Yaskawa INFORM job: DEMO_ROOF_UPPER_0625_3PAINT_57.JBI

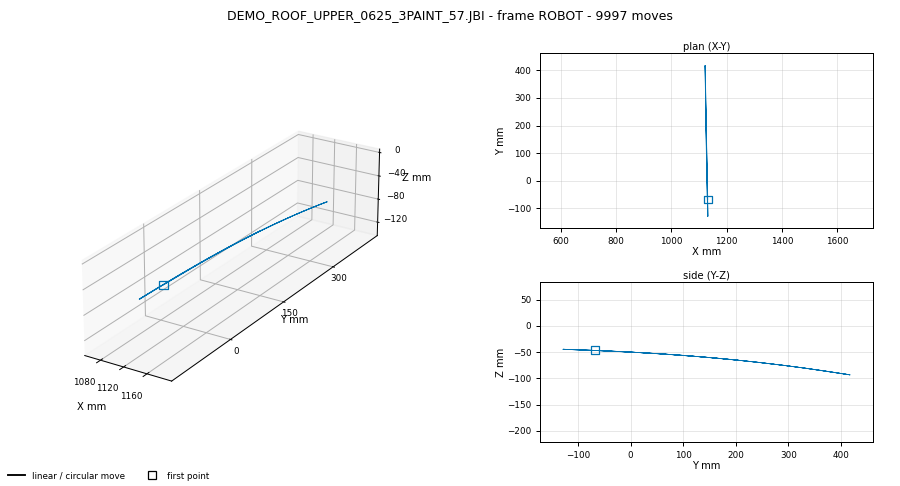
[picture p0: tool path of DEMO_ROOF_UPPER_0625_3PAINT_57.JBI in frame ROBOT, 9997 of 9997 moves have a stored position in this frame; points joined in program order, loops and branches not executed]
/JOB
//NAME DEMO_ROOF_UPPER_0625_3PAINT57
//POS
///NPOS 9997,0,0,0,0,0
///TOOL 0
///USER 0
///POSTYPE ROBOT
///RECTAN
///RCONF 1,0,0,0,0,0,0,0,0,0,0,0,0,0,0,0,0,0,0,0,0,0,0,0
C00000=1131.669,-67.518,-46.703,178.917,6.184,149.436
C00001=1131.665,-67.268,-46.713,178.919,6.185,149.435
C00002=1131.659,-67.019,-46.724,178.922,6.185,149.435
C00003=1131.653,-66.769,-46.734,178.924,6.186,149.434
C00004=1131.648,-66.519,-46.744,178.926,6.187,149.434
C00005=1131.643,-66.269,-46.754,178.928,6.187,149.433
C00006=1131.637,-66.020,-46.765,178.930,6.188,149.433
C00007=1131.632,-65.770,-46.775,178.932,6.188,149.432
C00008=1131.627,-65.520,-46.785,178.935,6.189,149.432
C00009=1131.622,-65.271,-46.795,178.937,6.189,149.431
C00010=1131.617,-65.021,-46.806,178.939,6.190,149.431
C00011=1131.611,-64.771,-46.816,178.941,6.190,149.430
C00012=1131.606,-64.521,-46.826,178.943,6.191,149.429
C00013=1131.601,-64.271,-46.837,178.946,6.191,149.429
C00014=1131.595,-64.022,-46.847,178.948,6.192,149.428
C00015=1131.590,-63.772,-46.858,178.950,6.193,149.428
C00016=1131.585,-63.522,-46.868,178.952,6.194,149.427
C00017=1131.579,-63.273,-46.879,178.955,6.194,149.427
C00018=1131.574,-63.023,-46.889,178.956,6.194,149.426
C00019=1131.568,-62.773,-46.899,178.959,6.195,149.426
C00020=1131.563,-62.524,-46.910,178.961,6.195,149.425
C00021=1131.558,-62.273,-46.920,178.963,6.196,149.425
C00022=1131.552,-62.024,-46.930,178.966,6.197,149.424
C00023=1131.548,-61.774,-46.940,178.968,6.197,149.424
C00024=1131.543,-61.525,-46.951,178.970,6.198,149.423
C00025=1131.537,-61.275,-46.961,178.972,6.198,149.423
C00026=1131.532,-61.025,-46.972,178.974,6.199,149.422
C00027=1131.527,-60.776,-46.982,178.976,6.199,149.421
C00028=1131.522,-60.525,-46.993,178.979,6.200,149.421
C00029=1131.516,-60.276,-47.004,178.981,6.201,149.421
C00030=1131.511,-60.026,-47.014,178.983,6.202,149.420
C00031=1131.506,-59.777,-47.025,178.985,6.202,149.420
C00032=1131.500,-59.527,-47.035,178.987,6.202,149.419
C00033=1131.495,-59.277,-47.045,178.989,6.203,149.418
C00034=1131.490,-59.028,-47.056,178.992,6.203,149.418
C00035=1131.485,-58.778,-47.067,178.994,6.204,149.417
C00036=1131.479,-58.528,-47.077,178.997,6.205,149.417
C00037=1131.474,-58.278,-47.088,178.999,6.205,149.416
C00038=1131.468,-58.029,-47.099,179.001,6.206,149.416
C00039=1131.463,-57.778,-47.110,179.003,6.207,149.415
C00040=1131.458,-57.529,-47.120,179.005,6.208,149.415
C00041=1131.453,-57.279,-47.130,179.007,6.207,149.414
C00042=1131.447,-57.030,-47.141,179.010,6.208,149.414
C00043=1131.442,-56.780,-47.152,179.012,6.209,149.413
C00044=1131.437,-56.530,-47.162,179.014,6.210,149.413
C00045=1131.431,-56.280,-47.172,179.016,6.210,149.412
C00046=1131.426,-56.031,-47.184,179.019,6.211,149.411
C00047=1131.421,-55.781,-47.194,179.021,6.211,149.411
C00048=1131.416,-55.531,-47.204,179.023,6.212,149.410
C00049=1131.410,-55.282,-47.215,179.025,6.213,149.410
C00050=1131.405,-55.032,-47.226,179.027,6.213,149.409
C00051=1131.400,-54.782,-47.236,179.030,6.213,149.409
C00052=1131.394,-54.532,-47.248,179.032,6.214,149.408
C00053=1131.389,-54.283,-47.258,179.034,6.215,149.408
C00054=1131.384,-54.033,-47.270,179.036,6.216,149.407
C00055=1131.379,-53.784,-47.280,179.039,6.216,149.407
C00056=1131.374,-53.533,-47.290,179.041,6.217,149.406
C00057=1131.369,-53.284,-47.302,179.043,6.218,149.406
C00058=1131.363,-53.034,-47.312,179.045,6.218,149.405
C00059=1131.358,-52.784,-47.324,179.048,6.219,149.405
C00060=1131.352,-52.535,-47.334,179.050,6.219,149.404
C00061=1131.347,-52.284,-47.345,179.052,6.219,149.404
C00062=1131.342,-52.036,-47.355,179.054,6.220,149.403
C00063=1131.337,-51.785,-47.366,179.057,6.221,149.402
C00064=1131.332,-51.536,-47.377,179.059,6.221,149.402
C00065=1131.326,-51.265,-47.388,179.061,6.222,149.401
C00066=1131.320,-50.994,-47.401,179.064,6.222,149.401
C00067=1131.314,-50.724,-47.413,179.066,6.223,149.400
C00068=1131.309,-50.453,-47.424,179.069,6.225,149.400
C00069=1131.303,-50.203,-47.435,179.071,6.224,149.399
C00070=1131.298,-49.953,-47.446,179.073,6.225,149.399
C00071=1131.293,-49.703,-47.457,179.075,6.226,149.398
C00072=1131.288,-49.454,-47.468,179.077,6.227,149.398
C00073=1131.282,-49.204,-47.479,179.080,6.227,149.397
C00074=1131.277,-48.955,-47.490,179.082,6.228,149.396
C00075=1131.272,-48.704,-47.501,179.084,6.229,149.396
C00076=1131.266,-48.456,-47.511,179.087,6.229,149.396
C00077=1131.261,-48.205,-47.523,179.089,6.230,149.395
C00078=1131.256,-47.955,-47.534,179.092,6.231,149.394
C00079=1131.250,-47.706,-47.544,179.094,6.231,149.394
C00080=1131.246,-47.456,-47.555,179.096,6.232,149.393
C00081=1131.240,-47.207,-47.567,179.099,6.232,149.393
C00082=1131.235,-46.957,-47.577,179.101,6.233,149.392
C00083=1131.230,-46.707,-47.589,179.103,6.234,149.392
C00084=1131.224,-46.457,-47.600,179.105,6.235,149.391
C00085=1131.219,-46.208,-47.611,179.108,6.235,149.391
C00086=1131.214,-45.958,-47.622,179.110,6.236,149.390
C00087=1131.208,-45.708,-47.633,179.112,6.236,149.390
C00088=1131.203,-45.459,-47.644,179.114,6.237,149.389
C00089=1131.198,-45.209,-47.654,179.116,6.237,149.388
C00090=1131.192,-44.959,-47.666,179.119,6.238,149.388
C00091=1131.188,-44.709,-47.678,179.121,6.239,149.387
C00092=1131.182,-44.460,-47.688,179.123,6.239,149.387
C00093=1131.176,-44.210,-47.700,179.126,6.240,149.386
C00094=1131.172,-43.960,-47.711,179.128,6.241,149.386
C00095=1131.166,-43.711,-47.721,179.130,6.241,149.385
C00096=1131.161,-43.461,-47.733,179.132,6.242,149.385
C00097=1131.156,-43.211,-47.744,179.135,6.243,149.384
C00098=1131.151,-42.962,-47.755,179.137,6.243,149.384
C00099=1131.145,-42.712,-47.767,179.139,6.244,149.383
C00100=1131.140,-42.462,-47.778,179.141,6.245,149.383
C00101=1131.134,-42.213,-47.789,179.144,6.245,149.382
C00102=1131.130,-41.963,-47.801,179.146,6.246,149.382
C00103=1131.125,-41.713,-47.811,179.149,6.247,149.381
C00104=1131.119,-41.463,-47.823,179.151,6.248,149.381
C00105=1131.114,-41.214,-47.834,179.153,6.248,149.380
C00106=1131.108,-40.964,-47.846,179.156,6.249,149.379
C00107=1131.103,-40.714,-47.856,179.158,6.249,149.379
C00108=1131.098,-40.465,-47.867,179.160,6.250,149.378
C00109=1131.093,-40.215,-47.879,179.163,6.251,149.378
C00110=1131.088,-39.965,-47.891,179.165,6.251,149.377
C00111=1131.082,-39.716,-47.902,179.167,6.252,149.377
C00112=1131.077,-39.466,-47.913,179.169,6.253,149.376
C00113=1131.072,-39.216,-47.925,179.172,6.253,149.376
C00114=1131.067,-38.966,-47.936,179.174,6.254,149.375
C00115=1131.061,-38.717,-47.947,179.176,6.255,149.375
C00116=1131.056,-38.468,-47.959,179.178,6.256,149.374
C00117=1131.051,-38.218,-47.971,179.181,6.256,149.373
C00118=1131.046,-37.967,-47.981,179.183,6.257,149.373
C00119=1131.040,-37.718,-47.993,179.185,6.258,149.373
C00120=1131.035,-37.469,-48.004,179.188,6.258,149.372
C00121=1131.030,-37.219,-48.016,179.190,6.259,149.371
C00122=1131.025,-36.969,-48.027,179.192,6.260,149.371
C00123=1131.019,-36.720,-48.039,179.195,6.260,149.370
C00124=1131.014,-36.470,-48.050,179.197,6.261,149.370
C00125=1131.009,-36.220,-48.062,179.200,6.262,149.369
C00126=1131.004,-35.971,-48.073,179.202,6.262,149.369
C00127=1130.998,-35.721,-48.085,179.204,6.263,149.368
C00128=1130.993,-35.471,-48.095,179.207,6.263,149.368
C00129=1130.988,-35.221,-48.107,179.209,6.264,149.367
C00130=1130.982,-34.971,-48.119,179.211,6.265,149.367
C00131=1130.977,-34.722,-48.130,179.213,6.266,149.366
C00132=1130.971,-34.472,-48.142,179.216,6.266,149.365
C00133=1130.967,-34.223,-48.153,179.218,6.267,149.365
C00134=1130.961,-33.973,-48.165,179.220,6.268,149.364
C00135=1130.957,-33.723,-48.176,179.223,6.268,149.364
C00136=1130.951,-33.473,-48.188,179.225,6.269,149.363
C00137=1130.945,-33.224,-48.200,179.227,6.270,149.363
C00138=1130.941,-32.974,-48.211,179.229,6.270,149.362
C00139=1130.935,-32.724,-48.223,179.232,6.271,149.362
C00140=1130.930,-32.475,-48.234,179.234,6.272,149.361
C00141=1130.925,-32.225,-48.246,179.236,6.272,149.361
C00142=1130.920,-31.975,-48.258,179.239,6.273,149.360
C00143=1130.915,-31.727,-48.269,179.242,6.274,149.360
C00144=1130.909,-31.477,-48.281,179.244,6.275,149.359
C00145=1130.904,-31.227,-48.293,179.246,6.276,149.359
C00146=1130.899,-30.977,-48.305,179.249,6.276,149.358
C00147=1130.894,-30.727,-48.316,179.251,6.277,149.357
C00148=1130.888,-30.477,-48.328,179.253,6.278,149.357
C00149=1130.883,-30.228,-48.340,179.255,6.279,149.356
C00150=1130.878,-29.978,-48.351,179.258,6.279,149.356
C00151=1130.872,-29.728,-48.363,179.260,6.280,149.355
C00152=1130.868,-29.479,-48.375,179.263,6.281,149.355
C00153=1130.862,-29.229,-48.387,179.265,6.281,149.354
C00154=1130.857,-28.980,-48.399,179.267,6.282,149.354
C00155=1130.852,-28.730,-48.410,179.270,6.283,149.353
C00156=1130.847,-28.480,-48.422,179.272,6.283,149.353
C00157=1130.841,-28.230,-48.434,179.274,6.284,149.352
C00158=1130.836,-27.980,-48.445,179.277,6.285,149.352
C00159=1130.831,-27.731,-48.458,179.279,6.285,149.351
C00160=1130.825,-27.482,-48.469,179.282,6.287,149.351
C00161=1130.820,-27.232,-48.481,179.284,6.287,149.350
C00162=1130.815,-26.982,-48.492,179.286,6.288,149.349
C00163=1130.810,-26.733,-48.505,179.289,6.289,149.349
C00164=1130.805,-26.483,-48.517,179.291,6.289,149.348
C00165=1130.800,-26.233,-48.528,179.293,6.290,149.348
C00166=1130.795,-25.983,-48.540,179.296,6.291,149.347
C00167=1130.789,-25.734,-48.553,179.298,6.292,149.347
C00168=1130.784,-25.484,-48.565,179.300,6.292,149.346
C00169=1130.779,-25.214,-48.578,179.303,6.293,149.346
C00170=1130.773,-24.944,-48.590,179.306,6.294,149.345
C00171=1130.767,-24.674,-48.603,179.308,6.295,149.344
C00172=1130.762,-24.404,-48.616,179.311,6.295,149.344
C00173=1130.756,-24.154,-48.628,179.313,6.296,149.343
C00174=1130.751,-23.904,-48.639,179.315,6.297,149.343
C00175=1130.746,-23.655,-48.652,179.318,6.297,149.342
C00176=1130.740,-23.405,-48.664,179.321,6.299,149.342
C00177=1130.735,-23.155,-48.675,179.323,6.299,149.341
C00178=1130.730,-22.906,-48.688,179.325,6.300,149.341
C00179=1130.725,-22.656,-48.700,179.328,6.301,149.340
C00180=1130.720,-22.407,-48.712,179.330,6.301,149.340
C00181=1130.714,-22.157,-48.724,179.332,6.302,149.339
C00182=1130.709,-21.907,-48.736,179.335,6.303,149.338
C00183=1130.704,-21.658,-48.749,179.337,6.303,149.338
C00184=1130.698,-21.408,-48.761,179.339,6.304,149.337
C00185=1130.694,-21.158,-48.772,179.342,6.306,149.337
C00186=1130.689,-20.909,-48.784,179.344,6.306,149.336
C00187=1130.683,-20.659,-48.796,179.347,6.307,149.336
C00188=1130.678,-20.410,-48.809,179.349,6.308,149.335
C00189=1130.673,-20.160,-48.821,179.352,6.308,149.335
C00190=1130.667,-19.910,-48.833,179.354,6.309,149.334
C00191=1130.662,-19.660,-48.845,179.356,6.310,149.334
C00192=1130.657,-19.411,-48.858,179.358,6.311,149.333
C00193=1130.651,-19.161,-48.870,179.361,6.311,149.332
C00194=1130.646,-18.912,-48.882,179.364,6.312,149.332
C00195=1130.642,-18.662,-48.894,179.366,6.313,149.332
C00196=1130.637,-18.412,-48.907,179.368,6.314,149.331
C00197=1130.632,-18.162,-48.919,179.371,6.314,149.330
C00198=1130.627,-17.913,-48.931,179.373,6.315,149.330
C00199=1130.621,-17.663,-48.943,179.375,6.316,149.329
C00200=1130.616,-17.414,-48.956,179.378,6.316,149.329
C00201=1130.611,-17.164,-48.968,179.380,6.318,149.328
C00202=1130.605,-16.914,-48.980,179.383,6.319,149.328
C00203=1130.600,-16.664,-48.992,179.385,6.319,149.327
C00204=1130.595,-16.415,-49.005,179.387,6.320,149.327
C00205=1130.589,-16.165,-49.017,179.390,6.321,149.326
C00206=1130.584,-15.916,-49.029,179.392,6.321,149.325
C00207=1130.579,-15.667,-49.042,179.394,6.322,149.325
C00208=1130.574,-15.417,-49.054,179.397,6.324,149.325
C00209=1130.569,-15.167,-49.067,179.399,6.324,149.324
C00210=1130.564,-14.917,-49.078,179.402,6.325,149.323
C00211=1130.559,-14.667,-49.091,179.404,6.326,149.323
C00212=1130.554,-14.418,-49.104,179.406,6.326,149.322
C00213=1130.548,-14.168,-49.116,179.409,6.327,149.322
C00214=1130.543,-13.919,-49.128,179.411,6.328,149.321
C00215=1130.538,-13.669,-49.141,179.414,6.329,149.321
C00216=1130.532,-13.420,-49.153,179.417,6.330,149.320
C00217=1130.527,-13.169,-49.166,179.419,6.330,149.320
C00218=1130.522,-12.920,-49.179,179.421,6.331,149.319
C00219=1130.517,-12.670,-49.191,179.423,6.332,149.319
C00220=1130.512,-12.421,-49.203,179.426,6.332,149.318
C00221=1130.506,-12.171,-49.216,179.429,6.334,149.318
C00222=1130.501,-11.921,-49.228,179.431,6.335,149.317
C00223=1130.496,-11.671,-49.241,179.434,6.335,149.316
C00224=1130.491,-11.422,-49.253,179.436,6.336,149.316
C00225=1130.486,-11.173,-49.266,179.438,6.337,149.315
C00226=1130.481,-10.923,-49.278,179.441,6.338,149.315
C00227=1130.476,-10.673,-49.290,179.443,6.339,149.314
C00228=1130.470,-10.424,-49.304,179.446,6.339,149.314
C00229=1130.465,-10.174,-49.317,179.448,6.340,149.313
C00230=1130.460,-9.924,-49.328,179.450,6.341,149.313
C00231=1130.455,-9.675,-49.341,179.453,6.341,149.312
C00232=1130.450,-9.425,-49.354,179.455,6.343,149.312
C00233=1130.444,-9.176,-49.366,179.458,6.343,149.311
C00234=1130.440,-8.926,-49.379,179.460,6.344,149.311
C00235=1130.434,-8.676,-49.392,179.462,6.345,149.310
C00236=1130.429,-8.426,-49.404,179.465,6.345,149.309
C00237=1130.424,-8.177,-49.417,179.468,6.347,149.309
C00238=1130.419,-7.927,-49.430,179.470,6.348,149.308
C00239=1130.414,-7.678,-49.442,179.472,6.349,149.308
C00240=1130.409,-7.428,-49.455,179.475,6.349,149.307
C00241=1130.403,-7.179,-49.468,179.477,6.350,149.307
C00242=1130.398,-6.929,-49.481,179.480,6.351,149.306
C00243=1130.393,-6.679,-49.493,179.482,6.352,149.306
C00244=1130.388,-6.429,-49.506,179.485,6.353,149.305
C00245=1130.382,-6.180,-49.519,179.487,6.353,149.305
C00246=1130.377,-5.931,-49.532,179.489,6.354,149.304
C00247=1130.372,-5.681,-49.544,179.492,6.355,149.304
C00248=1130.367,-5.431,-49.557,179.494,6.356,149.303
C00249=1130.361,-5.182,-49.570,179.497,6.357,149.302
C00250=1130.356,-4.932,-49.583,179.499,6.357,149.302
C00251=1130.352,-4.682,-49.596,179.502,6.359,149.301
C00252=1130.347,-4.433,-49.608,179.504,6.360,149.301
C00253=1130.341,-4.183,-49.622,179.507,6.360,149.300
C00254=1130.336,-3.933,-49.635,179.509,6.361,149.300
C00255=1130.331,-3.684,-49.647,179.511,6.362,149.299
C00256=1130.325,-3.434,-49.660,179.514,6.363,149.299
C00257=1130.321,-3.184,-49.673,179.517,6.364,149.298
C00258=1130.316,-2.935,-49.686,179.519,6.365,149.298
C00259=1130.310,-2.685,-49.699,179.521,6.365,149.297
C00260=1130.305,-2.436,-49.712,179.524,6.367,149.297
C00261=1130.300,-2.186,-49.725,179.526,6.367,149.296
C00262=1130.294,-1.936,-49.738,179.529,6.368,149.296
C00263=1130.289,-1.687,-49.751,179.531,6.369,149.295
C00264=1130.285,-1.437,-49.763,179.534,6.370,149.294
C00265=1130.279,-1.187,-49.777,179.536,6.371,149.294
C00266=1130.274,-0.938,-49.789,179.539,6.371,149.293
C00267=1130.269,-0.689,-49.803,179.541,6.372,149.293
C00268=1130.263,-0.439,-49.816,179.544,6.374,149.292
C00269=1130.258,-0.190,-49.829,179.547,6.374,149.292
C00270=1130.254,0.060,-49.842,179.549,6.375,149.291
C00271=1130.248,0.310,-49.855,179.551,6.376,149.291
C00272=1130.243,0.559,-49.868,179.554,6.377,149.290
C00273=1130.237,0.829,-49.882,179.556,6.378,149.290
C00274=1130.232,1.098,-49.896,179.559,6.379,149.289
C00275=1130.227,1.368,-49.910,179.562,6.380,149.288
C00276=1130.220,1.638,-49.924,179.564,6.381,149.288
C00277=1130.216,1.887,-49.938,179.567,6.382,149.287
C00278=1130.210,2.137,-49.951,179.569,6.383,149.287
C00279=1130.205,2.386,-49.964,179.572,6.383,149.286
C00280=1130.201,2.636,-49.977,179.575,6.385,149.286
C00281=1130.195,2.886,-49.990,179.577,6.385,149.285
C00282=1130.191,3.135,-50.004,179.579,6.386,149.285
C00283=1130.185,3.385,-50.017,179.582,6.387,149.284
C00284=1130.180,3.634,-50.030,179.585,6.388,149.284
C00285=1130.174,3.884,-50.043,179.587,6.389,149.283
C00286=1130.169,4.133,-50.056,179.589,6.389,149.282
C00287=1130.164,4.383,-50.070,179.592,6.390,149.282
C00288=1130.159,4.633,-50.083,179.594,6.392,149.282
C00289=1130.154,4.882,-50.097,179.597,6.393,149.281
C00290=1130.149,5.132,-50.109,179.599,6.393,149.280
C00291=1130.143,5.381,-50.123,179.602,6.395,149.280
C00292=1130.139,5.631,-50.136,179.604,6.395,149.279
C00293=1130.133,5.880,-50.150,179.607,6.396,149.279
C00294=1130.129,6.130,-50.162,179.610,6.397,149.278
C00295=1130.123,6.380,-50.176,179.612,6.398,149.278
C00296=1130.118,6.629,-50.189,179.614,6.399,149.277
C00297=1130.113,6.879,-50.203,179.617,6.399,149.277
C00298=1130.108,7.129,-50.217,179.619,6.401,149.276
C00299=1130.103,7.378,-50.229,179.622,6.402,149.276
C00300=1130.097,7.628,-50.243,179.624,6.402,149.275
C00301=1130.092,7.877,-50.256,179.627,6.404,149.275
C00302=1130.087,8.127,-50.270,179.629,6.405,149.274
C00303=1130.082,8.376,-50.283,179.632,6.405,149.273
C00304=1130.077,8.627,-50.297,179.635,6.407,149.273
C00305=1130.072,8.876,-50.311,179.637,6.408,149.273
C00306=1130.067,9.126,-50.324,179.639,6.408,149.272
C00307=1130.061,9.375,-50.337,179.642,6.410,149.271
C00308=1130.056,9.625,-50.351,179.644,6.410,149.271
C00309=1130.051,9.874,-50.364,179.647,6.411,149.270
C00310=1130.046,10.124,-50.378,179.649,6.412,149.270
C00311=1130.041,10.373,-50.391,179.652,6.413,149.269
C00312=1130.036,10.623,-50.405,179.654,6.414,149.269
C00313=1130.030,10.873,-50.418,179.657,6.414,149.268
C00314=1130.026,11.122,-50.432,179.660,6.416,149.268
C00315=1130.020,11.372,-50.445,179.662,6.417,149.267
C00316=1130.015,11.621,-50.459,179.664,6.417,149.267
C00317=1130.010,11.871,-50.472,179.667,6.419,149.266
C00318=1130.005,12.120,-50.486,179.669,6.420,149.266
C00319=1130.000,12.370,-50.500,179.672,6.420,149.265
C00320=1129.994,12.620,-50.514,179.675,6.422,149.264
C00321=1129.990,12.869,-50.527,179.677,6.422,149.264
C00322=1129.984,13.119,-50.540,179.680,6.424,149.264
C00323=1129.979,13.368,-50.555,179.682,6.424,149.263
C00324=1129.974,13.617,-50.568,179.685,6.425,149.262
C00325=1129.969,13.867,-50.582,179.687,6.427,149.262
C00326=1129.964,14.117,-50.596,179.690,6.427,149.261
C00327=1129.958,14.367,-50.609,179.692,6.428,149.261
C00328=1129.954,14.616,-50.623,179.695,6.430,149.260
C00329=1129.949,14.865,-50.637,179.698,6.430,149.260
C00330=1129.943,15.116,-50.650,179.700,6.431,149.259
C00331=1129.938,15.365,-50.664,179.703,6.433,149.259
C00332=1129.934,15.614,-50.678,179.705,6.433,149.258
C00333=1129.928,15.864,-50.691,179.707,6.434,149.258
C00334=1129.923,16.113,-50.705,179.710,6.435,149.257
C00335=1129.918,16.363,-50.720,179.712,6.436,149.257
C00336=1129.913,16.613,-50.734,179.716,6.437,149.256
C00337=1129.908,16.862,-50.746,179.718,6.438,149.256
C00338=1129.903,17.112,-50.761,179.720,6.439,149.255
C00339=1129.898,17.361,-50.775,179.723,6.440,149.254
C00340=1129.892,17.610,-50.789,179.725,6.441,149.254
C00341=1129.887,17.861,-50.802,179.728,6.442,149.253
C00342=1129.882,18.110,-50.817,179.731,6.443,149.253
C00343=1129.877,18.359,-50.830,179.733,6.444,149.252
C00344=1129.872,18.609,-50.844,179.736,6.446,149.252
C00345=1129.867,18.859,-50.858,179.738,6.446,149.251
C00346=1129.861,19.108,-50.872,179.741,6.447,149.251
C00347=1129.856,19.358,-50.886,179.743,6.448,149.250
C00348=1129.851,19.608,-50.900,179.746,6.449,149.250
C00349=1129.844,19.981,-50.921,179.750,6.451,149.249
C00350=1129.821,21.102,-50.984,179.631,6.695,149.338
C00351=1129.813,21.489,-51.006,179.634,6.702,149.338
C00352=1129.805,21.875,-51.028,179.635,6.709,149.339
C00353=1129.800,22.125,-51.042,179.635,6.714,149.340
C00354=1129.795,22.374,-51.056,179.637,6.718,149.341
C00355=1129.790,22.624,-51.070,179.638,6.723,149.342
C00356=1129.785,22.873,-51.085,179.639,6.727,149.342
C00357=1129.780,23.123,-51.099,179.640,6.732,149.343
C00358=1129.775,23.373,-51.113,179.641,6.736,149.344
C00359=1129.769,23.622,-51.127,179.642,6.740,149.344
C00360=1129.764,23.872,-51.141,179.643,6.745,149.345
C00361=1129.759,24.121,-51.156,179.644,6.749,149.346
C00362=1129.754,24.371,-51.170,179.646,6.755,149.346
C00363=1129.749,24.620,-51.184,179.647,6.759,149.347
C00364=1129.744,24.870,-51.198,179.648,6.763,149.348
C00365=1129.739,25.119,-51.212,179.649,6.768,149.348
C00366=1129.734,25.369,-51.227,179.650,6.772,149.349
C00367=1129.729,25.618,-51.242,179.651,6.776,149.350
C00368=1129.724,25.867,-51.255,179.652,6.781,149.350
C00369=1129.719,26.117,-51.270,179.654,6.786,149.351
C00370=1129.713,26.367,-51.285,179.655,6.790,149.352
C00371=1129.708,26.617,-51.299,179.656,6.794,149.352
C00372=1129.703,26.866,-51.313,179.657,6.799,149.353
C00373=1129.698,27.116,-51.327,179.658,6.803,149.353
C00374=1129.694,27.365,-51.342,179.659,6.807,149.354
C00375=1129.688,27.614,-51.356,179.660,6.812,149.355
C00376=1129.683,27.864,-51.371,179.662,6.817,149.355
C00377=1129.678,28.114,-51.385,179.663,6.821,149.356
C00378=1129.673,28.364,-51.400,179.664,6.825,149.357
C00379=1129.668,28.613,-51.415,179.665,6.830,149.357
C00380=1129.663,28.862,-51.429,179.666,6.834,149.358
C00381=1129.658,29.112,-51.443,179.667,6.838,149.359
C00382=1129.653,29.362,-51.458,179.668,6.843,149.359
C00383=1129.648,29.610,-51.472,179.669,6.847,149.360
C00384=1129.642,29.860,-51.487,179.670,6.851,149.361
C00385=1129.637,30.110,-51.501,179.672,6.856,149.361
C00386=1129.632,30.359,-51.516,179.673,6.861,149.362
C00387=1129.627,30.609,-51.531,179.674,6.865,149.363
C00388=1129.623,30.859,-51.545,179.675,6.869,149.363
C00389=1129.617,31.108,-51.561,179.676,6.874,149.364
C00390=1129.612,31.358,-51.575,179.678,6.877,149.364
C00391=1129.607,31.607,-51.589,179.679,6.882,149.365
C00392=1129.603,31.856,-51.604,179.680,6.886,149.366
C00393=1129.597,32.106,-51.619,179.681,6.890,149.366
C00394=1129.592,32.356,-51.634,179.682,6.895,149.367
C00395=1129.587,32.605,-51.648,179.683,6.900,149.367
C00396=1129.582,32.855,-51.663,179.684,6.904,149.368
C00397=1129.577,33.104,-51.678,179.686,6.908,149.369
C00398=1129.571,33.353,-51.692,179.687,6.913,149.369
C00399=1129.567,33.602,-51.707,179.688,6.917,149.370
C00400=1129.561,33.852,-51.722,179.689,6.921,149.370
C00401=1129.557,34.068,-51.735,179.690,6.925,149.371
C00402=1129.553,34.283,-51.748,179.691,6.928,149.372
C00403=1129.548,34.498,-51.760,179.692,6.933,149.372
C00404=1129.544,34.714,-51.773,179.693,6.936,149.373
C00405=1129.540,34.929,-51.786,179.695,6.940,149.373
C00406=1129.535,35.145,-51.798,179.695,6.943,149.374
C00407=1129.531,35.360,-51.812,179.697,6.947,149.374
C00408=1129.527,35.575,-51.824,179.697,6.951,149.375
C00409=1129.522,35.824,-51.840,179.699,6.955,149.375
C00410=1129.517,36.074,-51.854,179.700,6.959,149.376
C00411=1129.511,36.323,-51.870,179.701,6.963,149.377
C00412=1129.506,36.573,-51.884,179.702,6.968,149.377
C00413=1129.502,36.822,-51.899,179.703,6.972,149.378
C00414=1129.496,37.072,-51.914,179.705,6.977,149.378
C00415=1129.491,37.321,-51.929,179.706,6.981,149.379
C00416=1129.486,37.571,-51.944,179.707,6.985,149.380
C00417=1129.481,37.820,-51.959,179.708,6.990,149.380
C00418=1129.475,38.070,-51.974,179.710,6.994,149.381
C00419=1129.471,38.319,-51.989,179.711,6.998,149.381
C00420=1129.466,38.570,-52.005,179.712,7.002,149.382
C00421=1129.461,38.819,-52.020,179.713,7.006,149.383
C00422=1129.456,39.068,-52.035,179.715,7.010,149.383
C00423=1129.451,39.318,-52.049,179.716,7.015,149.384
C00424=1129.446,39.567,-52.064,179.717,7.019,149.384
C00425=1129.441,39.816,-52.080,179.718,7.023,149.385
C00426=1129.436,40.065,-52.095,179.719,7.027,149.385
C00427=1129.430,40.315,-52.110,179.720,7.032,149.386
C00428=1129.425,40.565,-52.125,179.722,7.036,149.387
C00429=1129.420,40.814,-52.140,179.723,7.040,149.387
C00430=1129.416,41.064,-52.156,179.724,7.044,149.388
C00431=1129.411,41.314,-52.171,179.725,7.048,149.388
C00432=1129.405,41.563,-52.186,179.727,7.052,149.389
C00433=1129.401,41.812,-52.201,179.728,7.057,149.389
C00434=1129.395,42.062,-52.217,179.730,7.062,149.390
C00435=1129.391,42.311,-52.232,179.731,7.066,149.390
C00436=1129.385,42.561,-52.247,179.732,7.070,149.391
C00437=1129.380,42.811,-52.263,179.733,7.074,149.392
C00438=1129.375,43.060,-52.278,179.735,7.078,149.392
C00439=1129.370,43.309,-52.293,179.736,7.082,149.393
C00440=1129.365,43.558,-52.308,179.737,7.087,149.393
C00441=1129.360,43.808,-52.324,179.738,7.091,149.394
C00442=1129.355,44.058,-52.340,179.740,7.095,149.395
C00443=1129.351,44.307,-52.355,179.741,7.099,149.395
C00444=1129.345,44.556,-52.370,179.742,7.103,149.396
C00445=1129.340,44.806,-52.386,179.743,7.108,149.396
C00446=1129.335,45.056,-52.400,179.745,7.111,149.397
C00447=1129.330,45.306,-52.416,179.746,7.116,149.397
C00448=1129.325,45.555,-52.431,179.747,7.120,149.398
C00449=1129.320,45.804,-52.447,179.749,7.124,149.398
C00450=1129.315,46.054,-52.462,179.750,7.128,149.399
C00451=1129.309,46.303,-52.478,179.751,7.132,149.399
C00452=1129.305,46.553,-52.493,179.752,7.136,149.400
C00453=1129.300,46.802,-52.509,179.754,7.140,149.401
C00454=1129.294,47.052,-52.524,179.755,7.145,149.401
C00455=1129.290,47.300,-52.540,179.756,7.149,149.402
C00456=1129.285,47.550,-52.556,179.757,7.153,149.402
C00457=1129.281,47.765,-52.569,179.759,7.157,149.403
C00458=1129.277,47.981,-52.582,179.760,7.160,149.403
C00459=1129.271,48.196,-52.596,179.761,7.164,149.404
C00460=1129.268,48.411,-52.610,179.762,7.167,149.404
C00461=1129.263,48.626,-52.623,179.763,7.171,149.405
C00462=1129.259,48.842,-52.636,179.764,7.174,149.405
C00463=1129.255,49.056,-52.650,179.765,7.178,149.405
C00464=1129.251,49.272,-52.664,179.766,7.182,149.406
C00465=1129.245,49.521,-52.679,179.768,7.186,149.407
C00466=1129.241,49.771,-52.695,179.769,7.190,149.407
C00467=1129.235,50.021,-52.711,179.771,7.194,149.408
C00468=1129.231,50.270,-52.726,179.772,7.198,149.408
C00469=1129.226,50.519,-52.742,179.773,7.202,149.409
C00470=1129.221,50.769,-52.758,179.774,7.207,149.409
C00471=1129.215,51.018,-52.773,179.776,7.210,149.410
C00472=1129.210,51.268,-52.789,179.777,7.215,149.410
C00473=1129.205,51.517,-52.806,179.779,7.219,149.411
C00474=1129.201,51.766,-52.821,179.780,7.223,149.411
C00475=1129.196,52.016,-52.837,179.781,7.227,149.412
C00476=1129.191,52.265,-52.852,179.783,7.231,149.412
C00477=1129.185,52.514,-52.869,179.784,7.235,149.413
C00478=1129.181,52.764,-52.885,179.785,7.239,149.413
C00479=1129.175,53.014,-52.900,179.787,7.243,149.414
C00480=1129.170,53.263,-52.916,179.788,7.247,149.414
C00481=1129.165,53.513,-52.932,179.789,7.252,149.415
C00482=1129.160,53.762,-52.948,179.791,7.255,149.415
C00483=1129.155,54.012,-52.964,179.792,7.260,149.416
C00484=1129.150,54.261,-52.980,179.793,7.264,149.417
C00485=1129.146,54.510,-52.995,179.794,7.268,149.417
C00486=1129.141,54.759,-53.012,179.796,7.272,149.418
C00487=1129.136,55.009,-53.027,179.798,7.276,149.418
C00488=1129.131,55.259,-53.043,179.799,7.280,149.419
C00489=1129.126,55.508,-53.060,179.800,7.284,149.419
C00490=1129.120,55.757,-53.075,179.801,7.288,149.420
C00491=1129.116,56.007,-53.092,179.803,7.292,149.420
C00492=1129.111,56.256,-53.108,179.804,7.297,149.421
C00493=1129.106,56.506,-53.124,179.806,7.300,149.421
C00494=1129.101,56.755,-53.140,179.807,7.304,149.422
C00495=1129.096,57.005,-53.156,179.808,7.309,149.422
C00496=1129.091,57.254,-53.172,179.810,7.313,149.423
C00497=1129.085,57.503,-53.188,179.811,7.317,149.423
C00498=1129.081,57.753,-53.204,179.812,7.321,149.424
C00499=1129.075,58.002,-53.221,179.814,7.325,149.424
C00500=1129.070,58.252,-53.237,179.815,7.329,149.425
C00501=1129.065,58.501,-53.253,179.817,7.333,149.425
C00502=1129.060,58.751,-53.269,179.818,7.337,149.426
C00503=1129.055,59.000,-53.286,179.819,7.341,149.426
C00504=1129.051,59.250,-53.302,179.821,7.345,149.427
C00505=1129.046,59.498,-53.318,179.822,7.349,149.427
C00506=1129.041,59.749,-53.334,179.824,7.353,149.428
C00507=1129.036,59.997,-53.350,179.825,7.357,149.428
C00508=1129.031,60.247,-53.366,179.826,7.361,149.429
C00509=1129.026,60.496,-53.383,179.828,7.365,149.429
C00510=1129.021,60.746,-53.400,179.828,7.369,149.430
C00511=1129.015,60.995,-53.415,179.830,7.373,149.430
C00512=1129.011,61.245,-53.432,179.831,7.377,149.431
C00513=1129.007,61.460,-53.446,179.833,7.381,149.431
C00514=1129.002,61.675,-53.460,179.834,7.384,149.432
C00515=1128.998,61.890,-53.474,179.835,7.388,149.432
C00516=1128.994,62.106,-53.488,179.836,7.391,149.433
C00517=1128.990,62.321,-53.503,179.838,7.395,149.433
C00518=1128.985,62.535,-53.517,179.839,7.398,149.433
C00519=1128.981,62.750,-53.531,179.840,7.401,149.434
C00520=1128.977,62.966,-53.546,179.841,7.405,149.434
C00521=1128.971,63.215,-53.561,179.843,7.409,149.435
C00522=1128.967,63.465,-53.578,179.844,7.413,149.435
C00523=1128.962,63.714,-53.595,179.846,7.417,149.436
C00524=1128.957,63.963,-53.611,179.847,7.421,149.436
C00525=1128.952,64.213,-53.627,179.848,7.425,149.437
C00526=1128.947,64.462,-53.644,179.850,7.429,149.437
C00527=1128.942,64.712,-53.660,179.851,7.433,149.438
C00528=1128.937,64.961,-53.678,179.853,7.437,149.438
C00529=1128.932,65.210,-53.694,179.854,7.441,149.439
C00530=1128.927,65.460,-53.711,179.855,7.445,149.439
C00531=1128.922,65.709,-53.726,179.857,7.449,149.440
C00532=1128.917,65.959,-53.743,179.858,7.453,149.440
C00533=1128.912,66.208,-53.760,179.860,7.457,149.441
C00534=1128.907,66.457,-53.776,179.861,7.461,149.441
C00535=1128.903,66.707,-53.793,179.863,7.465,149.442
C00536=1128.898,66.956,-53.810,179.864,7.469,149.442
C00537=1128.892,67.205,-53.827,179.865,7.473,149.443
C00538=1128.888,67.455,-53.843,179.866,7.477,149.443
C00539=1128.883,67.704,-53.861,179.868,7.481,149.444
C00540=1128.878,67.953,-53.877,179.869,7.485,149.444
C00541=1128.873,68.203,-53.894,179.871,7.489,149.445
C00542=1128.868,68.452,-53.911,179.872,7.493,149.445
C00543=1128.863,68.701,-53.927,179.874,7.497,149.446
C00544=1128.858,68.951,-53.944,179.875,7.501,149.446
C00545=1128.853,69.201,-53.961,179.876,7.505,149.447
C00546=1128.848,69.449,-53.977,179.878,7.509,149.447
C00547=1128.843,69.699,-53.995,179.880,7.513,149.448
C00548=1128.838,69.949,-54.011,179.881,7.517,149.448
C00549=1128.833,70.198,-54.029,179.882,7.521,149.449
C00550=1128.828,70.447,-54.045,179.884,7.525,149.449
C00551=1128.824,70.697,-54.062,179.885,7.529,149.450
C00552=1128.818,70.946,-54.079,179.886,7.533,149.450
C00553=1128.814,71.196,-54.095,179.888,7.537,149.451
C00554=1128.808,71.445,-54.112,179.890,7.541,149.451
C00555=1128.804,71.695,-54.129,179.891,7.545,149.452
C00556=1128.798,71.944,-54.146,179.892,7.549,149.452
C00557=1128.794,72.193,-54.164,179.894,7.553,149.452
C00558=1128.788,72.442,-54.181,179.895,7.557,149.453
C00559=1128.784,72.692,-54.197,179.897,7.561,149.453
C00560=1128.779,72.942,-54.214,179.898,7.565,149.454
C00561=1128.774,73.191,-54.231,179.900,7.569,149.454
C00562=1128.768,73.440,-54.248,179.901,7.573,149.455
C00563=1128.764,73.689,-54.265,179.902,7.577,149.455
C00564=1128.759,73.939,-54.283,179.904,7.581,149.456
C00565=1128.755,74.188,-54.299,179.906,7.585,149.456
C00566=1128.749,74.438,-54.317,179.907,7.589,149.457
C00567=1128.745,74.686,-54.334,179.908,7.593,149.457
C00568=1128.739,74.936,-54.351,179.910,7.597,149.458
C00569=1128.735,75.151,-54.366,179.911,7.600,149.458
C00570=1128.731,75.366,-54.381,179.912,7.604,149.459
C00571=1128.727,75.581,-54.395,179.913,7.607,149.459
C00572=1128.723,75.796,-54.410,179.915,7.610,149.459
C00573=1128.719,76.011,-54.425,179.916,7.614,149.460
C00574=1128.714,76.227,-54.440,179.917,7.617,149.460
C00575=1128.710,76.442,-54.454,179.919,7.621,149.461
C00576=1128.706,76.657,-54.470,179.920,7.624,149.461
C00577=1128.700,76.905,-54.486,179.921,7.628,149.462
C00578=1128.696,77.155,-54.504,179.922,7.631,149.462
C00579=1128.691,77.404,-54.521,179.922,7.635,149.463
C00580=1128.686,77.654,-54.538,179.924,7.639,149.463
C00581=1128.681,77.903,-54.556,179.925,7.642,149.464
C00582=1128.676,78.153,-54.573,179.926,7.646,149.464
C00583=1128.671,78.402,-54.590,179.927,7.649,149.465
C00584=1128.666,78.652,-54.608,179.928,7.654,149.465
C00585=1128.661,78.900,-54.624,179.929,7.657,149.466
C00586=1128.656,79.149,-54.642,179.930,7.661,149.467
C00587=1128.651,79.399,-54.659,179.931,7.664,149.467
C00588=1128.647,79.648,-54.677,179.932,7.669,149.468
C00589=1128.642,79.898,-54.694,179.933,7.672,149.468
C00590=1128.637,80.147,-54.712,179.934,7.676,149.469
C00591=1128.632,80.397,-54.729,179.935,7.679,149.469
C00592=1128.627,80.646,-54.747,179.936,7.683,149.470
C00593=1128.622,80.896,-54.764,179.938,7.687,149.470
C00594=1128.617,81.145,-54.782,179.938,7.691,149.471
C00595=1128.612,81.394,-54.798,179.940,7.695,149.471
C00596=1128.607,81.643,-54.816,179.940,7.698,149.472
C00597=1128.602,81.892,-54.834,179.942,7.702,149.472
C00598=1128.597,82.142,-54.852,179.943,7.706,149.473
C00599=1128.592,82.391,-54.869,179.944,7.709,149.473
C00600=1128.588,82.640,-54.886,179.946,7.713,149.474
C00601=1128.583,82.890,-54.903,179.947,7.718,149.474
C00602=1128.578,83.139,-54.921,179.948,7.721,149.475
C00603=1128.573,83.388,-54.939,179.949,7.725,149.476
C00604=1128.568,83.638,-54.956,179.950,7.729,149.476
C00605=1128.563,83.887,-54.974,179.951,7.732,149.476
C00606=1128.558,84.137,-54.991,179.952,7.736,149.477
C00607=1128.553,84.386,-55.009,179.954,7.740,149.477
C00608=1128.548,84.635,-55.027,179.955,7.744,149.478
C00609=1128.543,84.885,-55.045,179.956,7.748,149.478
C00610=1128.539,85.134,-55.062,179.958,7.751,149.479
C00611=1128.534,85.383,-55.080,179.959,7.756,149.480
C00612=1128.529,85.633,-55.097,179.961,7.760,149.480
C00613=1128.524,85.882,-55.115,179.962,7.764,149.480
C00614=1128.519,86.131,-55.133,179.963,7.767,149.481
C00615=1128.514,86.380,-55.151,179.964,7.771,149.481
C00616=1128.509,86.630,-55.168,179.966,7.775,149.482
C00617=1128.505,86.879,-55.186,179.967,7.779,149.482
C00618=1128.500,87.128,-55.204,179.969,7.783,149.483
C00619=1128.495,87.377,-55.222,179.970,7.787,149.483
C00620=1128.490,87.627,-55.239,179.971,7.790,149.484
C00621=1128.485,87.876,-55.257,179.973,7.794,149.484
C00622=1128.480,88.126,-55.275,179.974,7.798,149.485
C00623=1128.475,88.375,-55.293,179.975,7.802,149.485
C00624=1128.470,88.625,-55.310,179.977,7.806,149.486
C00625=1128.466,88.839,-55.326,179.978,7.809,149.486
C00626=1128.462,89.055,-55.341,179.980,7.813,149.487
C00627=1128.458,89.269,-55.357,179.981,7.816,149.487
C00628=1128.454,89.484,-55.372,179.983,7.820,149.487
C00629=1128.449,89.699,-55.388,179.984,7.823,149.488
C00630=1128.445,89.914,-55.403,179.985,7.826,149.488
C00631=1128.441,90.129,-55.419,179.986,7.830,149.489
C00632=1128.436,90.343,-55.434,179.987,7.833,149.489
C00633=1128.431,90.593,-55.451,179.989,7.837,149.489
C00634=1128.426,90.842,-55.469,179.990,7.841,149.490
C00635=1128.422,91.092,-55.488,179.992,7.844,149.490
C00636=1128.417,91.341,-55.506,179.993,7.848,149.491
C00637=1128.412,91.591,-55.524,179.995,7.852,149.491
C00638=1128.407,91.840,-55.542,179.997,7.856,149.492
C00639=1128.402,92.089,-55.560,179.998,7.860,149.492
C00640=1128.397,92.338,-55.578,180.000,7.864,149.492
C00641=1128.393,92.587,-55.596,-179.999,7.868,149.493
C00642=1128.388,92.836,-55.614,-179.997,7.872,149.493
C00643=1128.383,93.086,-55.632,-179.995,7.876,149.494
C00644=1128.378,93.336,-55.651,-179.993,7.880,149.494
C00645=1128.373,93.585,-55.669,-179.992,7.884,149.495
C00646=1128.368,93.834,-55.687,-179.990,7.888,149.495
C00647=1128.363,94.083,-55.705,-179.988,7.892,149.495
C00648=1128.358,94.333,-55.723,-179.987,7.896,149.496
C00649=1128.354,94.582,-55.741,-179.985,7.900,149.496
C00650=1128.349,94.831,-55.760,-179.984,7.904,149.497
C00651=1128.344,95.080,-55.778,-179.981,7.907,149.497
C00652=1128.339,95.330,-55.796,-179.979,7.912,149.497
C00653=1128.334,95.579,-55.814,-179.978,7.916,149.498
C00654=1128.329,95.829,-55.832,-179.976,7.920,149.498
C00655=1128.324,96.078,-55.850,-179.974,7.923,149.499
C00656=1128.320,96.327,-55.868,-179.973,7.927,149.499
C00657=1128.315,96.576,-55.887,-179.971,7.931,149.499
C00658=1128.310,96.826,-55.906,-179.969,7.936,149.500
C00659=1128.305,97.075,-55.924,-179.967,7.939,149.500
C00660=1128.300,97.324,-55.942,-179.965,7.943,149.501
C00661=1128.295,97.573,-55.961,-179.963,7.947,149.501
C00662=1128.290,97.823,-55.980,-179.961,7.951,149.501
C00663=1128.285,98.072,-55.998,-179.959,7.955,149.502
C00664=1128.281,98.321,-56.016,-179.958,7.959,149.502
C00665=1128.276,98.570,-56.034,-179.956,7.963,149.502
C00666=1128.271,98.820,-56.053,-179.954,7.967,149.503
C00667=1128.266,99.069,-56.071,-179.952,7.971,149.503
C00668=1128.261,99.318,-56.090,-179.950,7.975,149.503
C00669=1128.257,99.568,-56.108,-179.948,7.979,149.504
C00670=1128.251,99.817,-56.127,-179.946,7.983,149.504
C00671=1128.247,100.066,-56.146,-179.944,7.987,149.504
C00672=1128.242,100.315,-56.163,-179.942,7.990,149.505
C00673=1128.237,100.565,-56.182,-179.940,7.995,149.505
C00674=1128.232,100.814,-56.201,-179.938,7.999,149.505
C00675=1128.227,101.063,-56.219,-179.936,8.002,149.506
C00676=1128.223,101.312,-56.239,-179.934,8.007,149.506
C00677=1128.218,101.561,-56.257,-179.932,8.011,149.506
C00678=1128.212,101.811,-56.275,-179.930,8.015,149.507
C00679=1128.208,102.060,-56.294,-179.928,8.019,149.507
C00680=1128.203,102.309,-56.312,-179.925,8.022,149.507
C00681=1128.199,102.524,-56.329,-179.924,8.026,149.508
C00682=1128.195,102.739,-56.345,-179.922,8.030,149.508
C00683=1128.190,102.954,-56.362,-179.920,8.033,149.508
C00684=1128.186,103.168,-56.377,-179.918,8.037,149.508
C00685=1128.182,103.384,-56.394,-179.916,8.039,149.508
C00686=1128.178,103.598,-56.409,-179.915,8.043,149.509
C00687=1128.174,103.813,-56.426,-179.913,8.047,149.509
C00688=1128.170,104.028,-56.442,-179.911,8.050,149.509
C00689=1128.165,104.277,-56.461,-179.908,8.054,149.510
C00690=1128.161,104.527,-56.479,-179.906,8.058,149.510
C00691=1128.155,104.776,-56.499,-179.904,8.062,149.510
C00692=1128.151,105.024,-56.517,-179.901,8.066,149.510
C00693=1128.146,105.274,-56.536,-179.899,8.070,149.511
C00694=1128.141,105.523,-56.555,-179.897,8.074,149.511
C00695=1128.136,105.773,-56.575,-179.895,8.078,149.511
C00696=1128.131,106.022,-56.593,-179.892,8.082,149.511
C00697=1128.127,106.271,-56.612,-179.890,8.086,149.512
C00698=1128.122,106.520,-56.631,-179.888,8.090,149.512
C00699=1128.117,106.770,-56.650,-179.886,8.093,149.512
C00700=1128.112,107.019,-56.669,-179.883,8.098,149.512
C00701=1128.107,107.267,-56.688,-179.881,8.101,149.513
C00702=1128.102,107.517,-56.708,-179.879,8.106,149.513
C00703=1128.097,107.766,-56.726,-179.877,8.109,149.513
C00704=1128.093,108.016,-56.745,-179.874,8.114,149.513
C00705=1128.087,108.265,-56.765,-179.871,8.118,149.514
C00706=1128.083,108.514,-56.784,-179.869,8.121,149.514
C00707=1128.078,108.763,-56.803,-179.866,8.126,149.514
C00708=1128.074,109.013,-56.821,-179.864,8.129,149.514
C00709=1128.069,109.262,-56.841,-179.862,8.134,149.515
C00710=1128.063,109.511,-56.860,-179.859,8.137,149.515
C00711=1128.059,109.760,-56.879,-179.857,8.141,149.515
C00712=1128.054,110.009,-56.899,-179.854,8.145,149.515
C00713=1128.049,110.259,-56.918,-179.852,8.149,149.515
C00714=1128.045,110.507,-56.937,-179.849,8.153,149.515
C00715=1128.040,110.757,-56.957,-179.846,8.157,149.516
C00716=1128.035,111.006,-56.976,-179.844,8.161,149.516
C00717=1128.030,111.255,-56.995,-179.842,8.164,149.516
C00718=1128.026,111.505,-57.015,-179.840,8.168,149.516
C00719=1128.021,111.753,-57.034,-179.838,8.171,149.517
C00720=1128.016,112.003,-57.053,-179.837,8.175,149.517
C00721=1128.010,112.252,-57.073,-179.835,8.179,149.517
C00722=1128.006,112.501,-57.092,-179.832,8.182,149.517
C00723=1128.002,112.751,-57.112,-179.830,8.186,149.518
C00724=1127.996,113.000,-57.131,-179.828,8.189,149.518
C00725=1127.992,113.249,-57.150,-179.827,8.193,149.518
C00726=1127.986,113.498,-57.170,-179.825,8.197,149.519
C00727=1127.982,113.747,-57.189,-179.823,8.199,149.519
C00728=1127.978,113.997,-57.208,-179.821,8.203,149.519
C00729=1127.972,114.246,-57.228,-179.819,8.206,149.519
C00730=1127.967,114.495,-57.247,-179.817,8.210,149.520
C00731=1127.963,114.745,-57.267,-179.815,8.214,149.520
C00732=1127.958,114.993,-57.287,-179.813,8.217,149.520
C00733=1127.954,115.242,-57.306,-179.811,8.221,149.520
C00734=1127.949,115.492,-57.326,-179.809,8.224,149.520
C00735=1127.944,115.741,-57.345,-179.808,8.228,149.521
C00736=1127.939,115.990,-57.365,-179.806,8.232,149.521
C00737=1127.934,116.205,-57.381,-179.804,8.234,149.521
C00738=1127.930,116.420,-57.398,-179.803,8.237,149.522
C00739=1127.927,116.634,-57.416,-179.801,8.240,149.522
C00740=1127.922,116.849,-57.433,-179.799,8.243,149.522
C00741=1127.918,117.064,-57.450,-179.798,8.246,149.522
C00742=1127.914,117.278,-57.466,-179.796,8.249,149.522
C00743=1127.910,117.493,-57.483,-179.794,8.252,149.523
C00744=1127.906,117.708,-57.500,-179.793,8.255,149.523
C00745=1127.901,117.957,-57.520,-179.791,8.258,149.523
C00746=1127.897,118.206,-57.540,-179.789,8.262,149.523
C00747=1127.892,118.456,-57.560,-179.787,8.266,149.524
C00748=1127.887,118.705,-57.579,-179.785,8.269,149.524
C00749=1127.882,118.953,-57.599,-179.784,8.272,149.524
C00750=1127.877,119.203,-57.619,-179.781,8.275,149.524
C00751=1127.873,119.453,-57.639,-179.779,8.279,149.525
C00752=1127.868,119.701,-57.659,-179.778,8.283,149.525
C00753=1127.863,119.950,-57.678,-179.776,8.286,149.525
C00754=1127.858,120.199,-57.699,-179.774,8.289,149.526
C00755=1127.854,120.449,-57.718,-179.772,8.293,149.526
C00756=1127.848,120.698,-57.738,-179.770,8.296,149.526
C00757=1127.844,120.947,-57.758,-179.769,8.300,149.526
C00758=1127.839,121.196,-57.778,-179.766,8.303,149.527
C00759=1127.835,121.445,-57.798,-179.765,8.306,149.527
C00760=1127.829,121.694,-57.817,-179.763,8.310,149.527
C00761=1127.825,121.943,-57.838,-179.761,8.313,149.527
C00762=1127.820,122.193,-57.857,-179.759,8.317,149.528
C00763=1127.816,122.442,-57.878,-179.758,8.320,149.528
C00764=1127.810,122.692,-57.898,-179.756,8.323,149.528
C00765=1127.806,122.940,-57.918,-179.754,8.327,149.528
C00766=1127.800,123.189,-57.938,-179.752,8.330,149.529
C00767=1127.796,123.438,-57.958,-179.751,8.333,149.529
C00768=1127.791,123.688,-57.978,-179.749,8.337,149.529
C00769=1127.787,123.937,-57.998,-179.746,8.340,149.529
C00770=1127.782,124.186,-58.018,-179.744,8.344,149.530
C00771=1127.778,124.435,-58.038,-179.743,8.346,149.530
C00772=1127.772,124.684,-58.057,-179.741,8.350,149.530
C00773=1127.767,124.933,-58.078,-179.739,8.354,149.531
C00774=1127.763,125.182,-58.099,-179.738,8.357,149.531
C00775=1127.758,125.432,-58.118,-179.736,8.360,149.531
C00776=1127.754,125.681,-58.139,-179.734,8.364,149.531
C00777=1127.749,125.930,-58.159,-179.733,8.367,149.532
C00778=1127.744,126.179,-58.179,-179.731,8.370,149.532
C00779=1127.739,126.429,-58.200,-179.729,8.374,149.532
C00780=1127.734,126.677,-58.220,-179.728,8.377,149.533
C00781=1127.729,126.926,-58.239,-179.725,8.380,149.533
C00782=1127.725,127.175,-58.260,-179.723,8.384,149.533
C00783=1127.721,127.424,-58.280,-179.721,8.387,149.533
C00784=1127.715,127.674,-58.300,-179.720,8.390,149.534
C00785=1127.711,127.923,-58.321,-179.718,8.394,149.534
C00786=1127.706,128.172,-58.341,-179.717,8.397,149.534
C00787=1127.702,128.421,-58.361,-179.715,8.400,149.534
C00788=1127.696,128.671,-58.382,-179.713,8.404,149.535
C00789=1127.692,128.920,-58.402,-179.712,8.407,149.535
C00790=1127.687,129.169,-58.422,-179.710,8.410,149.535
C00791=1127.682,129.418,-58.443,-179.708,8.414,149.535
C00792=1127.677,129.667,-58.463,-179.707,8.417,149.536
C00793=1127.673,129.882,-58.480,-179.705,8.419,149.536
C00794=1127.670,130.096,-58.498,-179.703,8.423,149.536
C00795=1127.665,130.311,-58.516,-179.702,8.426,149.537
C00796=1127.661,130.525,-58.533,-179.700,8.428,149.537
C00797=1127.657,130.740,-58.551,-179.699,8.431,149.537
C00798=1127.653,130.955,-58.568,-179.697,8.434,149.537
C00799=1127.649,131.170,-58.586,-179.696,8.437,149.538
C00800=1127.645,131.384,-58.604,-179.695,8.440,149.538
C00801=1127.641,131.633,-58.625,-179.693,8.443,149.538
C00802=1127.635,131.882,-58.646,-179.691,8.446,149.538
C00803=1127.630,132.131,-58.666,-179.690,8.450,149.539
C00804=1127.626,132.380,-58.685,-179.688,8.453,149.539
C00805=1127.620,132.629,-58.706,-179.686,8.456,149.539
C00806=1127.616,132.878,-58.727,-179.685,8.460,149.540
C00807=1127.611,133.128,-58.748,-179.683,8.462,149.540
C00808=1127.607,133.377,-58.768,-179.681,8.466,149.540
C00809=1127.603,133.626,-58.789,-179.679,8.470,149.541
C00810=1127.597,133.876,-58.810,-179.678,8.473,149.541
C00811=1127.593,134.124,-58.830,-179.676,8.476,149.541
C00812=1127.588,134.374,-58.851,-179.675,8.479,149.541
C00813=1127.583,134.623,-58.871,-179.673,8.483,149.542
C00814=1127.578,134.872,-58.892,-179.671,8.485,149.542
C00815=1127.574,135.121,-58.913,-179.670,8.489,149.542
C00816=1127.569,135.370,-58.933,-179.668,8.492,149.543
C00817=1127.564,135.619,-58.954,-179.667,8.496,149.543
C00818=1127.560,135.867,-58.975,-179.665,8.499,149.543
C00819=1127.555,136.117,-58.996,-179.663,8.502,149.543
C00820=1127.550,136.366,-59.016,-179.661,8.506,149.544
C00821=1127.545,136.615,-59.037,-179.660,8.509,149.544
C00822=1127.541,136.864,-59.058,-179.658,8.512,149.544
C00823=1127.536,137.113,-59.079,-179.657,8.515,149.545
C00824=1127.531,137.362,-59.099,-179.655,8.519,149.545
C00825=1127.526,137.611,-59.120,-179.654,8.522,149.545
C00826=1127.522,137.861,-59.141,-179.652,8.525,149.546
C00827=1127.517,138.110,-59.162,-179.651,8.528,149.546
C00828=1127.513,138.359,-59.183,-179.649,8.532,149.546
C00829=1127.508,138.608,-59.204,-179.648,8.535,149.547
C00830=1127.502,138.857,-59.225,-179.646,8.538,149.547
C00831=1127.498,139.106,-59.245,-179.645,8.541,149.547
C00832=1127.493,139.355,-59.267,-179.643,8.545,149.548
C00833=1127.489,139.604,-59.287,-179.642,8.548,149.548
C00834=1127.484,139.854,-59.309,-179.639,8.552,149.548
C00835=1127.480,140.103,-59.329,-179.638,8.555,149.549
C00836=1127.475,140.351,-59.351,-179.636,8.558,149.549
C00837=1127.470,140.600,-59.372,-179.635,8.561,149.549
C00838=1127.465,140.849,-59.392,-179.633,8.565,149.550
C00839=1127.460,141.099,-59.413,-179.632,8.568,149.550
C00840=1127.456,141.347,-59.434,-179.631,8.572,149.550
C00841=1127.451,141.597,-59.455,-179.629,8.574,149.551
C00842=1127.446,141.846,-59.476,-179.628,8.578,149.551
C00843=1127.442,142.095,-59.497,-179.626,8.581,149.551
C00844=1127.437,142.344,-59.518,-179.624,8.585,149.552
C00845=1127.432,142.593,-59.539,-179.623,8.588,149.552
C00846=1127.428,142.842,-59.561,-179.621,8.591,149.552
C00847=1127.423,143.091,-59.582,-179.620,8.594,149.553
C00848=1127.418,143.341,-59.603,-179.618,8.598,149.553
C00849=1127.414,143.554,-59.621,-179.617,8.601,149.553
C00850=1127.410,143.769,-59.640,-179.616,8.604,149.554
C00851=1127.406,143.984,-59.657,-179.614,8.606,149.554
C00852=1127.402,144.199,-59.676,-179.613,8.610,149.554
C00853=1127.398,144.413,-59.694,-179.612,8.612,149.555
C00854=1127.394,144.627,-59.713,-179.611,8.615,149.555
C00855=1127.390,144.842,-59.731,-179.610,8.617,149.555
C00856=1127.386,145.057,-59.749,-179.609,8.620,149.556
C00857=1127.381,145.306,-59.770,-179.606,8.624,149.556
C00858=1127.376,145.554,-59.791,-179.603,8.629,149.556
C00859=1127.372,145.803,-59.812,-179.600,8.633,149.556
C00860=1127.367,146.052,-59.833,-179.598,8.636,149.556
C00861=1127.362,146.302,-59.855,-179.596,8.641,149.557
C00862=1127.357,146.551,-59.876,-179.593,8.644,149.557
C00863=1127.353,146.799,-59.898,-179.590,8.649,149.557
C00864=1127.349,147.049,-59.919,-179.588,8.652,149.557
C00865=1127.344,147.298,-59.941,-179.585,8.656,149.557
C00866=1127.339,147.547,-59.962,-179.582,8.660,149.557
C00867=1127.334,147.795,-59.983,-179.580,8.664,149.558
C00868=1127.330,148.045,-60.005,-179.577,8.668,149.558
C00869=1127.324,148.294,-60.026,-179.575,8.671,149.558
C00870=1127.320,148.542,-60.047,-179.572,8.675,149.558
C00871=1127.316,148.792,-60.069,-179.569,8.680,149.558
C00872=1127.311,149.041,-60.090,-179.567,8.683,149.558
C00873=1127.306,149.290,-60.112,-179.564,8.687,149.559
C00874=1127.302,149.539,-60.134,-179.562,8.691,149.559
C00875=1127.296,149.788,-60.155,-179.559,8.694,149.559
C00876=1127.292,150.037,-60.177,-179.556,8.699,149.559
C00877=1127.287,150.286,-60.199,-179.553,8.702,149.559
C00878=1127.282,150.535,-60.220,-179.551,8.706,149.559
C00879=1127.277,150.784,-60.241,-179.549,8.710,149.560
C00880=1127.273,151.033,-60.263,-179.545,8.714,149.560
C00881=1127.268,151.282,-60.285,-179.543,8.717,149.560
C00882=1127.263,151.531,-60.307,-179.540,8.721,149.560
C00883=1127.259,151.780,-60.329,-179.538,8.724,149.560
C00884=1127.254,152.029,-60.350,-179.535,8.728,149.560
C00885=1127.250,152.279,-60.372,-179.533,8.732,149.560
C00886=1127.245,152.527,-60.394,-179.530,8.735,149.560
C00887=1127.240,152.776,-60.415,-179.528,8.739,149.561
C00888=1127.236,153.025,-60.437,-179.526,8.743,149.561
C00889=1127.231,153.274,-60.459,-179.522,8.746,149.561
C00890=1127.226,153.523,-60.481,-179.520,8.750,149.561
C00891=1127.222,153.772,-60.503,-179.517,8.754,149.561
C00892=1127.217,154.021,-60.525,-179.515,8.757,149.561
C00893=1127.212,154.270,-60.546,-179.513,8.760,149.561
C00894=1127.208,154.519,-60.568,-179.509,8.764,149.561
C00895=1127.203,154.768,-60.590,-179.507,8.768,149.562
C00896=1127.198,155.017,-60.612,-179.505,8.771,149.562
C00897=1127.194,155.266,-60.634,-179.502,8.775,149.562
C00898=1127.189,155.515,-60.656,-179.500,8.778,149.562
C00899=1127.184,155.764,-60.678,-179.498,8.782,149.562
C00900=1127.179,156.013,-60.700,-179.494,8.786,149.562
C00901=1127.175,156.262,-60.722,-179.492,8.789,149.562
C00902=1127.170,156.511,-60.744,-179.490,8.792,149.563
C00903=1127.166,156.760,-60.766,-179.487,8.796,149.563
C00904=1127.160,157.009,-60.788,-179.485,8.800,149.563
C00905=1127.158,157.224,-60.807,-179.483,8.802,149.563
C00906=1127.154,157.438,-60.826,-179.480,8.805,149.563
C00907=1127.149,157.652,-60.845,-179.478,8.809,149.563
C00908=1127.145,157.866,-60.864,-179.476,8.811,149.563
C00909=1127.141,158.080,-60.883,-179.474,8.814,149.563
C00910=1127.138,158.296,-60.902,-179.472,8.817,149.563
C00911=1127.133,158.510,-60.921,-179.470,8.820,149.563
C00912=1127.129,158.724,-60.940,-179.467,8.823,149.563
C00913=1127.124,158.974,-60.963,-179.465,8.826,149.564
C00914=1127.120,159.222,-60.985,-179.463,8.830,149.564
C00915=1127.116,159.471,-61.007,-179.459,8.833,149.564
C00916=1127.110,159.720,-61.029,-179.457,8.837,149.564
C00917=1127.106,159.969,-61.052,-179.455,8.840,149.564
C00918=1127.102,160.218,-61.074,-179.452,8.843,149.564
C00919=1127.097,160.467,-61.096,-179.450,8.847,149.564
C00920=1127.092,160.717,-61.119,-179.448,8.850,149.564
C00921=1127.087,160.965,-61.141,-179.445,8.853,149.564
C00922=1127.083,161.214,-61.163,-179.443,8.856,149.565
C00923=1127.078,161.463,-61.186,-179.440,8.860,149.565
C00924=1127.073,161.712,-61.208,-179.437,8.863,149.565
C00925=1127.069,161.961,-61.230,-179.435,8.866,149.565
C00926=1127.064,162.209,-61.253,-179.433,8.870,149.565
C00927=1127.060,162.459,-61.275,-179.430,8.873,149.565
C00928=1127.056,162.707,-61.298,-179.428,8.876,149.565
C00929=1127.050,162.956,-61.320,-179.426,8.880,149.565
C00930=1127.046,163.206,-61.342,-179.423,8.883,149.565
C00931=1127.041,163.455,-61.366,-179.421,8.886,149.565
C00932=1127.036,163.703,-61.387,-179.418,8.889,149.566
C00933=1127.032,163.952,-61.410,-179.416,8.892,149.566
C00934=1127.027,164.202,-61.433,-179.413,8.895,149.566
C00935=1127.023,164.450,-61.455,-179.411,8.899,149.566
C00936=1127.018,164.699,-61.478,-179.409,8.902,149.566
C00937=1127.014,164.948,-61.501,-179.406,8.905,149.566
C00938=1127.009,165.197,-61.524,-179.404,8.908,149.566
C00939=1127.004,165.446,-61.546,-179.401,8.911,149.566
C00940=1126.999,165.695,-61.569,-179.399,8.915,149.566
C00941=1126.995,165.944,-61.591,-179.397,8.918,149.566
C00942=1126.990,166.193,-61.614,-179.394,8.921,149.566
C00943=1126.986,166.441,-61.637,-179.392,8.924,149.566
C00944=1126.981,166.691,-61.659,-179.390,8.928,149.567
C00945=1126.977,166.940,-61.682,-179.387,8.931,149.567
C00946=1126.972,167.188,-61.705,-179.384,8.934,149.567
C00947=1126.967,167.437,-61.727,-179.382,8.937,149.567
C00948=1126.963,167.686,-61.751,-179.380,8.940,149.567
C00949=1126.959,167.935,-61.773,-179.378,8.943,149.567
C00950=1126.953,168.184,-61.796,-179.375,8.946,149.567
C00951=1126.948,168.433,-61.819,-179.373,8.949,149.567
C00952=1126.944,168.682,-61.842,-179.371,8.953,149.567
C00953=1126.939,168.931,-61.864,-179.368,8.956,149.567
C00954=1126.935,169.180,-61.887,-179.366,8.959,149.567
C00955=1126.930,169.428,-61.910,-179.364,8.962,149.568
C00956=1126.925,169.677,-61.933,-179.362,8.965,149.568
C00957=1126.921,169.926,-61.956,-179.359,8.968,149.568
C00958=1126.916,170.176,-61.979,-179.357,8.971,149.568
C00959=1126.912,170.425,-62.002,-179.355,8.974,149.568
C00960=1126.907,170.673,-62.025,-179.352,8.977,149.568
C00961=1126.903,170.888,-62.045,-179.350,8.980,149.568
C00962=1126.899,171.102,-62.064,-179.348,8.982,149.568
C00963=1126.896,171.317,-62.084,-179.347,8.985,149.568
C00964=1126.891,171.530,-62.104,-179.344,8.988,149.568
C00965=1126.887,171.745,-62.123,-179.342,8.990,149.568
C00966=1126.884,171.959,-62.144,-179.341,8.992,149.568
C00967=1126.879,172.173,-62.163,-179.339,8.995,149.568
C00968=1126.876,172.388,-62.183,-179.337,8.998,149.569
C00969=1126.871,172.637,-62.207,-179.335,9.001,149.569
C00970=1126.866,172.885,-62.230,-179.332,9.004,149.569
C00971=1126.862,173.134,-62.253,-179.330,9.007,149.569
C00972=1126.857,173.383,-62.276,-179.328,9.010,149.569
C00973=1126.853,173.632,-62.299,-179.326,9.013,149.569
C00974=1126.848,173.881,-62.323,-179.323,9.016,149.569
C00975=1126.844,174.130,-62.345,-179.321,9.019,149.569
C00976=1126.839,174.379,-62.369,-179.319,9.022,149.569
C00977=1126.835,174.628,-62.392,-179.317,9.025,149.569
C00978=1126.830,174.877,-62.415,-179.315,9.028,149.569
C00979=1126.825,175.125,-62.438,-179.312,9.031,149.570
C00980=1126.821,175.374,-62.461,-179.310,9.034,149.570
C00981=1126.816,175.623,-62.485,-179.308,9.037,149.570
C00982=1126.811,175.872,-62.508,-179.305,9.040,149.570
C00983=1126.806,176.121,-62.531,-179.304,9.043,149.570
C00984=1126.802,176.370,-62.555,-179.301,9.046,149.570
C00985=1126.798,176.619,-62.577,-179.299,9.049,149.570
C00986=1126.793,176.867,-62.601,-179.297,9.051,149.570
C00987=1126.789,177.116,-62.625,-179.295,9.055,149.570
C00988=1126.784,177.365,-62.648,-179.293,9.057,149.570
C00989=1126.779,177.614,-62.672,-179.291,9.060,149.570
C00990=1126.775,177.863,-62.695,-179.288,9.063,149.571
C00991=1126.770,178.112,-62.718,-179.287,9.066,149.571
C00992=1126.766,178.361,-62.742,-179.284,9.069,149.571
C00993=1126.762,178.609,-62.765,-179.282,9.072,149.571
C00994=1126.757,178.858,-62.788,-179.280,9.075,149.571
C00995=1126.752,179.107,-62.812,-179.278,9.078,149.571
C00996=1126.747,179.356,-62.835,-179.275,9.081,149.571
C00997=1126.743,179.605,-62.859,-179.273,9.084,149.571
C00998=1126.738,179.854,-62.883,-179.269,9.088,149.571
C00999=1126.734,180.103,-62.906,-179.266,9.091,149.571
C01000=1126.729,180.351,-62.930,-179.263,9.095,149.571
C01001=1126.725,180.600,-62.953,-179.261,9.098,149.571
C01002=1126.720,180.849,-62.977,-179.258,9.102,149.571
C01003=1126.715,181.098,-63.001,-179.255,9.105,149.571
C01004=1126.711,181.347,-63.024,-179.251,9.109,149.571
C01005=1126.706,181.596,-63.048,-179.249,9.112,149.571
C01006=1126.702,181.844,-63.072,-179.246,9.114,149.571
C01007=1126.697,182.093,-63.095,-179.243,9.117,149.571
C01008=1126.693,182.342,-63.119,-179.240,9.121,149.571
C01009=1126.688,182.591,-63.142,-179.238,9.124,149.571
C01010=1126.683,182.840,-63.166,-179.235,9.127,149.571
C01011=1126.679,183.088,-63.190,-179.232,9.130,149.571
C01012=1126.675,183.338,-63.214,-179.230,9.133,149.571
C01013=1126.670,183.586,-63.238,-179.227,9.137,149.571
C01014=1126.666,183.835,-63.261,-179.224,9.140,149.571
C01015=1126.661,184.084,-63.285,-179.221,9.143,149.571
C01016=1126.656,184.333,-63.308,-179.219,9.146,149.571
C01017=1126.653,184.547,-63.330,-179.217,9.149,149.571
C01018=1126.648,184.761,-63.350,-179.214,9.152,149.571
C01019=1126.644,184.975,-63.371,-179.212,9.154,149.571
C01020=1126.641,185.189,-63.391,-179.210,9.156,149.571
C01021=1126.637,185.403,-63.412,-179.207,9.159,149.571
C01022=1126.633,185.618,-63.432,-179.206,9.161,149.571
C01023=1126.629,185.833,-63.453,-179.204,9.164,149.571
C01024=1126.624,186.046,-63.474,-179.201,9.167,149.571
C01025=1126.620,186.295,-63.498,-179.199,9.170,149.571
C01026=1126.616,186.544,-63.522,-179.197,9.172,149.571
C01027=1126.612,186.793,-63.545,-179.194,9.175,149.571
C01028=1126.607,187.041,-63.570,-179.191,9.178,149.571
C01029=1126.602,187.290,-63.594,-179.189,9.181,149.571
C01030=1126.597,187.539,-63.618,-179.187,9.184,149.571
C01031=1126.593,187.788,-63.642,-179.184,9.187,149.571
C01032=1126.589,188.037,-63.666,-179.182,9.190,149.571
C01033=1126.584,188.286,-63.690,-179.180,9.192,149.571
C01034=1126.579,188.534,-63.714,-179.177,9.195,149.571
C01035=1126.575,188.783,-63.738,-179.175,9.198,149.571
C01036=1126.570,189.031,-63.762,-179.173,9.201,149.571
C01037=1126.566,189.281,-63.787,-179.170,9.204,149.571
C01038=1126.561,189.530,-63.811,-179.169,9.206,149.571
C01039=1126.557,189.778,-63.835,-179.166,9.209,149.572
C01040=1126.552,190.027,-63.859,-179.164,9.212,149.572
C01041=1126.547,190.275,-63.883,-179.163,9.214,149.572
C01042=1126.544,190.524,-63.908,-179.160,9.217,149.572
C01043=1126.539,190.773,-63.931,-179.158,9.220,149.572
C01044=1126.534,191.022,-63.956,-179.156,9.223,149.572
C01045=1126.529,191.271,-63.980,-179.154,9.225,149.572
C01046=1126.526,191.520,-64.004,-179.152,9.227,149.572
C01047=1126.520,191.768,-64.029,-179.150,9.231,149.572
C01048=1126.516,192.017,-64.053,-179.148,9.233,149.572
C01049=1126.511,192.265,-64.078,-179.146,9.236,149.572
C01050=1126.507,192.515,-64.102,-179.145,9.238,149.573
C01051=1126.502,192.764,-64.126,-179.142,9.241,149.573
C01052=1126.497,193.012,-64.150,-179.140,9.244,149.573
C01053=1126.493,193.261,-64.175,-179.139,9.246,149.573
C01054=1126.489,193.510,-64.199,-179.137,9.249,149.573
C01055=1126.484,193.759,-64.224,-179.135,9.251,149.573
C01056=1126.480,194.007,-64.248,-179.133,9.254,149.573
C01057=1126.475,194.256,-64.273,-179.131,9.256,149.573
C01058=1126.471,194.505,-64.297,-179.129,9.260,149.573
C01059=1126.465,194.754,-64.321,-179.127,9.262,149.573
C01060=1126.462,195.003,-64.346,-179.126,9.265,149.574
C01061=1126.457,195.251,-64.370,-179.125,9.267,149.574
C01062=1126.452,195.500,-64.395,-179.123,9.270,149.574
C01063=1126.448,195.749,-64.419,-179.121,9.272,149.574
C01064=1126.443,195.998,-64.444,-179.120,9.275,149.574
C01065=1126.439,196.246,-64.468,-179.118,9.277,149.575
C01066=1126.435,196.495,-64.493,-179.115,9.281,149.575
C01067=1126.430,196.743,-64.518,-179.111,9.285,149.574
C01068=1126.425,196.992,-64.542,-179.108,9.288,149.574
C01069=1126.421,197.241,-64.567,-179.104,9.292,149.574
C01070=1126.416,197.490,-64.591,-179.100,9.295,149.574
C01071=1126.412,197.738,-64.615,-179.096,9.300,149.574
C01072=1126.407,197.988,-64.640,-179.093,9.303,149.574
C01073=1126.404,198.202,-64.662,-179.090,9.306,149.574
C01074=1126.400,198.416,-64.683,-179.087,9.309,149.574
C01075=1126.396,198.630,-64.704,-179.083,9.313,149.574
C01076=1126.392,198.843,-64.725,-179.081,9.315,149.573
C01077=1126.388,199.057,-64.747,-179.078,9.318,149.573
C01078=1126.385,199.271,-64.768,-179.075,9.321,149.573
C01079=1126.380,199.486,-64.790,-179.071,9.324,149.573
C01080=1126.376,199.700,-64.811,-179.069,9.327,149.573
C01081=1126.372,199.949,-64.835,-179.065,9.331,149.573
C01082=1126.368,200.197,-64.861,-179.062,9.334,149.573
C01083=1126.363,200.446,-64.886,-179.058,9.337,149.573
C01084=1126.359,200.695,-64.910,-179.055,9.341,149.572
C01085=1126.354,200.943,-64.935,-179.052,9.343,149.572
C01086=1126.350,201.193,-64.960,-179.048,9.347,149.572
C01087=1126.345,201.441,-64.985,-179.045,9.350,149.572
C01088=1126.341,201.690,-65.010,-179.042,9.353,149.572
C01089=1126.336,201.939,-65.035,-179.038,9.357,149.572
C01090=1126.332,202.187,-65.060,-179.035,9.359,149.572
C01091=1126.327,202.436,-65.085,-179.032,9.362,149.571
C01092=1126.323,202.685,-65.111,-179.029,9.366,149.571
C01093=1126.318,202.934,-65.135,-179.026,9.368,149.571
C01094=1126.314,203.182,-65.160,-179.023,9.371,149.571
C01095=1126.309,203.431,-65.185,-179.020,9.375,149.571
C01096=1126.305,203.680,-65.211,-179.017,9.378,149.571
C01097=1126.300,203.928,-65.236,-179.014,9.381,149.571
C01098=1126.296,204.177,-65.261,-179.011,9.383,149.571
C01099=1126.292,204.425,-65.286,-179.007,9.387,149.570
C01100=1126.287,204.674,-65.311,-179.005,9.390,149.571
C01101=1126.282,204.922,-65.336,-179.002,9.393,149.570
C01102=1126.278,205.171,-65.362,-178.999,9.395,149.570
C01103=1126.273,205.421,-65.387,-178.996,9.398,149.570
C01104=1126.269,205.669,-65.413,-178.993,9.401,149.570
C01105=1126.265,205.918,-65.437,-178.990,9.404,149.570
C01106=1126.260,206.166,-65.462,-178.987,9.407,149.570
C01107=1126.256,206.415,-65.488,-178.985,9.410,149.570
C01108=1126.251,206.663,-65.514,-178.982,9.413,149.570
C01109=1126.246,206.912,-65.539,-178.980,9.415,149.570
C01110=1126.242,207.161,-65.564,-178.977,9.418,149.570
C01111=1126.237,207.409,-65.590,-178.974,9.420,149.569
C01112=1126.233,207.658,-65.615,-178.972,9.423,149.570
C01113=1126.229,207.907,-65.640,-178.970,9.426,149.570
C01114=1126.224,208.156,-65.666,-178.967,9.429,149.569
C01115=1126.220,208.404,-65.692,-178.964,9.432,149.570
C01116=1126.215,208.652,-65.717,-178.962,9.434,149.569
C01117=1126.210,208.902,-65.742,-178.959,9.437,149.569
C01118=1126.207,209.150,-65.767,-178.957,9.440,149.569
C01119=1126.202,209.398,-65.793,-178.955,9.442,149.570
C01120=1126.198,209.647,-65.818,-178.952,9.445,149.569
C01121=1126.193,209.896,-65.844,-178.950,9.447,149.569
C01122=1126.189,210.144,-65.869,-178.948,9.450,149.569
C01123=1126.184,210.393,-65.895,-178.946,9.453,149.570
C01124=1126.180,210.642,-65.921,-178.943,9.456,149.570
C01125=1126.175,210.890,-65.946,-178.941,9.458,149.570
C01126=1126.170,211.140,-65.972,-178.939,9.460,149.570
C01127=1126.166,211.388,-65.998,-178.937,9.464,149.570
C01128=1126.162,211.637,-66.023,-178.935,9.466,149.570
C01129=1126.158,211.851,-66.046,-178.933,9.468,149.570
C01130=1126.154,212.065,-66.068,-178.932,9.471,149.570
C01131=1126.150,212.279,-66.089,-178.930,9.473,149.570
C01132=1126.146,212.492,-66.112,-178.928,9.475,149.570
C01133=1126.143,212.706,-66.133,-178.926,9.477,149.570
C01134=1126.138,212.921,-66.156,-178.925,9.480,149.570
C01135=1126.135,213.134,-66.178,-178.923,9.482,149.570
C01136=1126.131,213.348,-66.200,-178.922,9.484,149.571
C01137=1126.126,213.597,-66.226,-178.920,9.487,149.571
C01138=1126.122,213.846,-66.251,-178.918,9.490,149.571
C01139=1126.118,214.095,-66.277,-178.916,9.492,149.571
C01140=1126.113,214.343,-66.302,-178.915,9.495,149.571
C01141=1126.109,214.591,-66.329,-178.912,9.498,149.571
C01142=1126.105,214.840,-66.355,-178.911,9.500,149.571
C01143=1126.100,215.089,-66.381,-178.909,9.503,149.572
C01144=1126.095,215.337,-66.406,-178.907,9.506,149.572
C01145=1126.091,215.586,-66.432,-178.905,9.509,149.572
C01146=1126.087,215.835,-66.458,-178.903,9.512,149.572
C01147=1126.083,216.083,-66.484,-178.901,9.514,149.572
C01148=1126.078,216.332,-66.509,-178.899,9.518,149.572
C01149=1126.073,216.580,-66.536,-178.897,9.520,149.572
C01150=1126.069,216.829,-66.562,-178.894,9.523,149.572
C01151=1126.065,217.078,-66.588,-178.892,9.527,149.573
C01152=1126.060,217.326,-66.613,-178.890,9.529,149.573
C01153=1126.056,217.575,-66.639,-178.888,9.532,149.573
C01154=1126.051,217.824,-66.665,-178.885,9.536,149.573
C01155=1126.047,218.072,-66.692,-178.883,9.539,149.573
C01156=1126.042,218.321,-66.717,-178.881,9.541,149.573
C01157=1126.038,218.569,-66.743,-178.879,9.544,149.573
C01158=1126.033,218.819,-66.769,-178.876,9.547,149.573
C01159=1126.029,219.066,-66.796,-178.874,9.551,149.574
C01160=1126.025,219.315,-66.821,-178.871,9.554,149.574
C01161=1126.020,219.564,-66.847,-178.869,9.557,149.574
C01162=1126.016,219.812,-66.874,-178.866,9.560,149.574
C01163=1126.011,220.061,-66.900,-178.864,9.562,149.574
C01164=1126.007,220.310,-66.926,-178.862,9.565,149.574
C01165=1126.003,220.558,-66.952,-178.859,9.569,149.574
C01166=1125.998,220.806,-66.978,-178.856,9.572,149.574
C01167=1125.994,221.055,-67.004,-178.854,9.576,149.574
C01168=1125.990,221.303,-67.030,-178.851,9.579,149.574
C01169=1125.985,221.552,-67.057,-178.849,9.582,149.574
C01170=1125.981,221.801,-67.083,-178.846,9.585,149.574
C01171=1125.976,222.050,-67.109,-178.844,9.588,149.574
C01172=1125.972,222.298,-67.136,-178.841,9.591,149.574
C01173=1125.968,222.547,-67.162,-178.838,9.595,149.574
C01174=1125.963,222.796,-67.188,-178.835,9.598,149.574
C01175=1125.959,223.044,-67.214,-178.833,9.601,149.575
C01176=1125.953,223.292,-67.240,-178.830,9.604,149.575
C01177=1125.949,223.541,-67.267,-178.827,9.608,149.574
C01178=1125.945,223.789,-67.293,-178.824,9.611,149.575
C01179=1125.940,224.038,-67.320,-178.822,9.614,149.575
C01180=1125.936,224.286,-67.346,-178.818,9.618,149.575
C01181=1125.931,224.535,-67.373,-178.816,9.621,149.575
C01182=1125.928,224.783,-67.399,-178.812,9.625,149.575
C01183=1125.923,225.033,-67.425,-178.809,9.627,149.575
C01184=1125.919,225.281,-67.452,-178.807,9.630,149.575
C01185=1125.915,225.494,-67.475,-178.804,9.633,149.574
C01186=1125.911,225.709,-67.498,-178.801,9.636,149.575
C01187=1125.907,225.922,-67.521,-178.799,9.639,149.575
C01188=1125.903,226.136,-67.543,-178.796,9.642,149.574
C01189=1125.900,226.350,-67.566,-178.793,9.645,149.575
C01190=1125.896,226.564,-67.589,-178.790,9.648,149.574
C01191=1125.892,226.777,-67.611,-178.788,9.651,149.574
C01192=1125.889,226.992,-67.635,-178.785,9.654,149.574
C01193=1125.884,227.240,-67.662,-178.781,9.657,149.574
C01194=1125.880,227.489,-67.689,-178.778,9.660,149.574
C01195=1125.875,227.738,-67.714,-178.775,9.664,149.574
C01196=1125.871,227.986,-67.742,-178.772,9.668,149.574
C01197=1125.867,228.234,-67.768,-178.769,9.670,149.574
C01198=1125.862,228.483,-67.795,-178.765,9.674,149.574
C01199=1125.857,228.731,-67.822,-178.762,9.677,149.574
C01200=1125.853,228.980,-67.848,-178.758,9.681,149.574
C01201=1125.849,229.228,-67.875,-178.754,9.684,149.573
C01202=1125.845,229.477,-67.901,-178.751,9.687,149.573
C01203=1125.840,229.725,-67.928,-178.748,9.691,149.573
C01204=1125.835,229.974,-67.956,-178.744,9.694,149.573
C01205=1125.831,230.222,-67.983,-178.741,9.698,149.573
C01206=1125.827,230.471,-68.009,-178.737,9.701,149.573
C01207=1125.823,230.720,-68.036,-178.733,9.704,149.573
C01208=1125.818,230.968,-68.064,-178.730,9.707,149.572
C01209=1125.814,231.216,-68.090,-178.727,9.711,149.572
C01210=1125.809,231.465,-68.117,-178.723,9.714,149.572
C01211=1125.805,231.713,-68.144,-178.720,9.717,149.572
C01212=1125.800,231.962,-68.171,-178.717,9.720,149.572
C01213=1125.797,232.211,-68.198,-178.714,9.723,149.572
C01214=1125.792,232.459,-68.225,-178.711,9.726,149.572
C01215=1125.788,232.708,-68.252,-178.707,9.729,149.572
C01216=1125.783,232.956,-68.279,-178.704,9.732,149.571
C01217=1125.778,233.205,-68.306,-178.701,9.736,149.571
C01218=1125.775,233.452,-68.333,-178.697,9.738,149.571
C01219=1125.771,233.701,-68.361,-178.694,9.741,149.571
C01220=1125.766,233.950,-68.388,-178.691,9.744,149.571
C01221=1125.761,234.198,-68.415,-178.688,9.746,149.571
C01222=1125.757,234.447,-68.442,-178.685,9.750,149.571
C01223=1125.752,234.695,-68.470,-178.682,9.753,149.570
C01224=1125.748,234.944,-68.497,-178.679,9.755,149.570
C01225=1125.744,235.192,-68.524,-178.676,9.758,149.570
C01226=1125.740,235.441,-68.551,-178.673,9.761,149.570
C01227=1125.735,235.688,-68.579,-178.670,9.764,149.570
C01228=1125.731,235.938,-68.606,-178.667,9.767,149.570
C01229=1125.727,236.186,-68.633,-178.665,9.769,149.570
C01230=1125.722,236.435,-68.660,-178.662,9.771,149.570
C01231=1125.718,236.683,-68.688,-178.659,9.774,149.570
C01232=1125.713,236.932,-68.715,-178.656,9.777,149.569
C01233=1125.709,237.180,-68.742,-178.653,9.780,149.569
C01234=1125.704,237.428,-68.770,-178.650,9.782,149.569
C01235=1125.700,237.677,-68.798,-178.649,9.785,149.569
C01236=1125.696,237.925,-68.825,-178.646,9.788,149.569
C01237=1125.691,238.174,-68.852,-178.643,9.790,149.569
C01238=1125.687,238.422,-68.879,-178.640,9.792,149.569
C01239=1125.683,238.671,-68.908,-178.638,9.795,149.569
C01240=1125.678,238.919,-68.935,-178.635,9.797,149.569
C01241=1125.675,239.133,-68.959,-178.634,9.800,149.569
C01242=1125.671,239.346,-68.982,-178.631,9.802,149.569
C01243=1125.667,239.561,-69.006,-178.629,9.804,149.569
C01244=1125.664,239.774,-69.029,-178.627,9.806,149.569
C01245=1125.660,239.987,-69.053,-178.625,9.808,149.569
C01246=1125.656,240.201,-69.077,-178.623,9.810,149.569
C01247=1125.653,240.415,-69.100,-178.621,9.813,149.569
C01248=1125.649,240.628,-69.124,-178.619,9.815,149.568
C01249=1125.644,240.878,-69.152,-178.617,9.817,149.569
C01250=1125.640,241.126,-69.180,-178.614,9.819,149.568
C01251=1125.636,241.374,-69.208,-178.612,9.822,149.568
C01252=1125.631,241.623,-69.235,-178.610,9.824,149.569
C01253=1125.627,241.870,-69.263,-178.608,9.826,149.568
C01254=1125.623,242.120,-69.290,-178.606,9.829,149.568
C01255=1125.618,242.368,-69.318,-178.604,9.831,149.569
C01256=1125.614,242.616,-69.345,-178.602,9.833,149.568
C01257=1125.610,242.865,-69.373,-178.600,9.835,149.568
C01258=1125.605,243.113,-69.402,-178.598,9.838,149.568
C01259=1125.601,243.362,-69.429,-178.596,9.840,149.569
C01260=1125.597,243.610,-69.457,-178.594,9.842,149.569
C01261=1125.592,243.858,-69.485,-178.592,9.845,149.569
C01262=1125.588,244.107,-69.512,-178.590,9.847,149.569
C01263=1125.584,244.355,-69.540,-178.588,9.849,149.569
C01264=1125.580,244.603,-69.568,-178.586,9.852,149.569
C01265=1125.575,244.852,-69.596,-178.585,9.854,149.569
C01266=1125.570,245.100,-69.623,-178.583,9.856,149.569
C01267=1125.567,245.349,-69.651,-178.582,9.858,149.569
C01268=1125.562,245.597,-69.678,-178.580,9.860,149.569
C01269=1125.558,245.846,-69.707,-178.578,9.863,149.569
C01270=1125.553,246.094,-69.735,-178.576,9.865,149.569
C01271=1125.549,246.342,-69.763,-178.575,9.867,149.570
C01272=1125.545,246.591,-69.790,-178.573,9.869,149.570
C01273=1125.540,246.839,-69.818,-178.572,9.872,149.570
C01274=1125.536,247.088,-69.847,-178.571,9.874,149.570
C01275=1125.531,247.336,-69.875,-178.569,9.876,149.570
C01276=1125.527,247.585,-69.902,-178.565,9.880,149.570
C01277=1125.523,247.833,-69.930,-178.558,9.885,149.569
C01278=1125.519,248.082,-69.958,-178.553,9.890,149.569
C01279=1125.514,248.329,-69.986,-178.546,9.895,149.569
C01280=1125.510,248.578,-70.014,-178.541,9.899,149.568
C01281=1125.505,248.826,-70.043,-178.535,9.904,149.568
C01282=1125.502,249.075,-70.071,-178.529,9.908,149.567
C01283=1125.497,249.323,-70.099,-178.524,9.913,149.567
C01284=1125.493,249.572,-70.127,-178.519,9.916,149.567
C01285=1125.488,249.819,-70.155,-178.514,9.920,149.566
C01286=1125.485,250.068,-70.183,-178.509,9.924,149.566
C01287=1125.480,250.316,-70.212,-178.505,9.928,149.566
C01288=1125.476,250.565,-70.240,-178.501,9.931,149.565
C01289=1125.471,250.813,-70.268,-178.497,9.934,149.565
C01290=1125.467,251.062,-70.296,-178.493,9.937,149.565
C01291=1125.463,251.310,-70.325,-178.489,9.940,149.564
C01292=1125.458,251.558,-70.353,-178.485,9.943,149.564
C01293=1125.454,251.807,-70.382,-178.482,9.945,149.564
C01294=1125.450,252.054,-70.410,-178.479,9.948,149.564
C01295=1125.446,252.303,-70.438,-178.476,9.951,149.563
C01296=1125.441,252.552,-70.467,-178.474,9.953,149.563
C01297=1125.437,252.765,-70.492,-178.471,9.955,149.563
C01298=1125.434,252.978,-70.516,-178.469,9.957,149.563
C01299=1125.430,253.192,-70.540,-178.468,9.958,149.563
C01300=1125.427,253.406,-70.565,-178.466,9.960,149.563
C01301=1125.423,253.620,-70.590,-178.464,9.962,149.563
C01302=1125.419,253.832,-70.614,-178.463,9.963,149.563
C01303=1125.416,254.046,-70.638,-178.461,9.965,149.563
C01304=1125.412,254.260,-70.663,-178.460,9.966,149.563
C01305=1125.407,254.509,-70.692,-178.460,9.967,149.563
C01306=1125.403,254.756,-70.720,-178.459,9.969,149.563
C01307=1125.399,255.005,-70.749,-178.458,9.970,149.563
C01308=1125.395,255.254,-70.777,-178.458,9.972,149.564
C01309=1125.390,255.502,-70.806,-178.458,9.972,149.564
C01310=1125.386,255.750,-70.834,-178.458,9.973,149.564
C01311=1125.382,255.999,-70.863,-178.458,9.974,149.564
C01312=1125.377,256.247,-70.892,-178.455,9.978,149.564
C01313=1125.373,256.495,-70.920,-178.452,9.980,149.564
C01314=1125.369,256.744,-70.949,-178.449,9.983,149.564
C01315=1125.365,256.991,-70.977,-178.446,9.986,149.564
C01316=1125.360,257.240,-71.006,-178.443,9.989,149.564
C01317=1125.356,257.489,-71.035,-178.440,9.991,149.564
C01318=1125.352,257.736,-71.063,-178.437,9.994,149.564
C01319=1125.347,257.985,-71.092,-178.434,9.998,149.564
C01320=1125.344,258.233,-71.121,-178.431,10.001,149.564
C01321=1125.339,258.481,-71.149,-178.428,10.004,149.564
C01322=1125.334,258.730,-71.178,-178.425,10.006,149.564
C01323=1125.331,258.978,-71.207,-178.422,10.009,149.563
C01324=1125.326,259.226,-71.235,-178.419,10.013,149.563
C01325=1125.322,259.475,-71.265,-178.415,10.015,149.563
C01326=1125.318,259.723,-71.293,-178.413,10.018,149.563
C01327=1125.314,259.971,-71.322,-178.409,10.021,149.563
C01328=1125.309,260.220,-71.351,-178.406,10.024,149.563
C01329=1125.304,260.468,-71.380,-178.403,10.027,149.563
C01330=1125.301,260.716,-71.409,-178.400,10.030,149.563
C01331=1125.296,260.965,-71.438,-178.396,10.033,149.562
C01332=1125.292,261.213,-71.467,-178.393,10.036,149.562
C01333=1125.287,261.461,-71.496,-178.390,10.039,149.562
C01334=1125.284,261.709,-71.525,-178.386,10.042,149.562
C01335=1125.280,261.957,-71.554,-178.383,10.045,149.562
C01336=1125.275,262.206,-71.583,-178.379,10.048,149.561
C01337=1125.270,262.454,-71.612,-178.376,10.051,149.561
C01338=1125.266,262.702,-71.641,-178.372,10.054,149.561
C01339=1125.262,262.951,-71.670,-178.369,10.057,149.561
C01340=1125.258,263.199,-71.699,-178.365,10.060,149.561
C01341=1125.254,263.447,-71.728,-178.361,10.063,149.560
C01342=1125.250,263.696,-71.758,-178.358,10.066,149.560
C01343=1125.245,263.944,-71.786,-178.354,10.069,149.560
C01344=1125.241,264.192,-71.816,-178.350,10.073,149.560
C01345=1125.236,264.440,-71.845,-178.347,10.075,149.560
C01346=1125.232,264.689,-71.874,-178.344,10.078,149.559
C01347=1125.228,264.937,-71.904,-178.342,10.080,149.559
C01348=1125.223,265.186,-71.933,-178.339,10.083,149.559
C01349=1125.219,265.433,-71.962,-178.337,10.084,149.559
C01350=1125.215,265.681,-71.991,-178.334,10.087,149.559
C01351=1125.211,265.929,-72.020,-178.331,10.089,149.559
C01352=1125.207,266.178,-72.050,-178.328,10.092,149.559
C01353=1125.203,266.391,-72.075,-178.326,10.094,149.559
C01354=1125.199,266.605,-72.100,-178.324,10.096,149.559
C01355=1125.195,266.818,-72.126,-178.322,10.098,149.559
C01356=1125.192,267.032,-72.151,-178.320,10.100,149.558
C01357=1125.188,267.245,-72.176,-178.318,10.103,149.558
C01358=1125.185,267.459,-72.201,-178.315,10.105,149.558
C01359=1125.181,267.672,-72.226,-178.313,10.107,149.558
C01360=1125.178,267.885,-72.252,-178.311,10.109,149.558
C01361=1125.173,268.134,-72.281,-178.308,10.111,149.558
C01362=1125.169,268.382,-72.310,-178.305,10.113,149.558
C01363=1125.165,268.630,-72.340,-178.303,10.116,149.558
C01364=1125.161,268.879,-72.369,-178.300,10.119,149.558
C01365=1125.157,269.127,-72.399,-178.297,10.121,149.558
C01366=1125.152,269.375,-72.429,-178.294,10.124,149.557
C01367=1125.148,269.624,-72.458,-178.291,10.126,149.557
C01368=1125.143,269.872,-72.488,-178.288,10.129,149.557
C01369=1125.139,270.120,-72.517,-178.286,10.131,149.557
C01370=1125.135,270.368,-72.547,-178.283,10.134,149.557
C01371=1125.131,270.616,-72.577,-178.280,10.137,149.557
C01372=1125.127,270.864,-72.606,-178.277,10.139,149.557
C01373=1125.123,271.113,-72.636,-178.275,10.141,149.557
C01374=1125.119,271.361,-72.665,-178.272,10.144,149.557
C01375=1125.114,271.609,-72.695,-178.269,10.147,149.556
C01376=1125.110,271.858,-72.725,-178.266,10.150,149.556
C01377=1125.106,272.105,-72.755,-178.263,10.152,149.556
C01378=1125.102,272.354,-72.784,-178.260,10.155,149.556
C01379=1125.097,272.602,-72.814,-178.257,10.158,149.556
C01380=1125.093,272.850,-72.843,-178.255,10.160,149.556
C01381=1125.089,273.098,-72.873,-178.252,10.163,149.556
C01382=1125.084,273.346,-72.903,-178.249,10.165,149.556
C01383=1125.080,273.595,-72.933,-178.246,10.168,149.555
C01384=1125.076,273.843,-72.962,-178.243,10.171,149.555
C01385=1125.072,274.091,-72.993,-178.240,10.173,149.555
C01386=1125.068,274.339,-73.022,-178.237,10.176,149.555
C01387=1125.063,274.587,-73.052,-178.234,10.179,149.555
C01388=1125.059,274.835,-73.082,-178.231,10.182,149.555
C01389=1125.055,275.083,-73.112,-178.228,10.184,149.555
C01390=1125.051,275.332,-73.141,-178.225,10.187,149.555
C01391=1125.046,275.580,-73.172,-178.222,10.189,149.554
C01392=1125.042,275.828,-73.201,-178.219,10.192,149.554
C01393=1125.038,276.075,-73.232,-178.215,10.195,149.554
C01394=1125.035,276.324,-73.261,-178.212,10.198,149.554
C01395=1125.030,276.572,-73.292,-178.209,10.201,149.554
C01396=1125.026,276.821,-73.322,-178.206,10.203,149.554
C01397=1125.022,277.069,-73.351,-178.203,10.206,149.554
C01398=1125.017,277.317,-73.382,-178.200,10.209,149.553
C01399=1125.013,277.565,-73.411,-178.197,10.211,149.553
C01400=1125.009,277.813,-73.441,-178.193,10.215,149.553
C01401=1125.005,278.061,-73.473,-178.190,10.217,149.553
C01402=1125.001,278.310,-73.502,-178.187,10.220,149.553
C01403=1124.997,278.557,-73.532,-178.183,10.222,149.552
C01404=1124.992,278.806,-73.562,-178.180,10.225,149.552
C01405=1124.988,279.054,-73.592,-178.176,10.228,149.552
C01406=1124.983,279.302,-73.622,-178.174,10.231,149.552
C01407=1124.980,279.551,-73.653,-178.170,10.234,149.552
C01408=1124.976,279.798,-73.683,-178.167,10.236,149.552
C01409=1124.972,280.012,-73.709,-178.164,10.239,149.551
C01410=1124.968,280.225,-73.735,-178.161,10.241,149.551
C01411=1124.964,280.438,-73.761,-178.158,10.244,149.551
C01412=1124.961,280.652,-73.787,-178.155,10.246,149.551
C01413=1124.957,280.865,-73.813,-178.152,10.249,149.551
C01414=1124.953,281.078,-73.840,-178.149,10.251,149.550
C01415=1124.950,281.292,-73.865,-178.147,10.253,149.550
C01416=1124.946,281.505,-73.891,-178.143,10.255,149.550
C01417=1124.943,281.753,-73.922,-178.140,10.258,149.550
C01418=1124.938,282.001,-73.953,-178.137,10.261,149.550
C01419=1124.934,282.249,-73.983,-178.134,10.263,149.550
C01420=1124.929,282.497,-74.013,-178.131,10.266,149.549
C01421=1124.926,282.746,-74.044,-178.128,10.269,149.549
C01422=1124.921,282.994,-74.074,-178.125,10.271,149.549
C01423=1124.917,283.241,-74.104,-178.122,10.273,149.549
C01424=1124.913,283.489,-74.135,-178.119,10.276,149.549
C01425=1124.909,283.738,-74.166,-178.116,10.279,149.549
C01426=1124.905,283.986,-74.196,-178.113,10.281,149.548
C01427=1124.900,284.234,-74.227,-178.110,10.284,149.548
C01428=1124.897,284.482,-74.257,-178.107,10.286,149.548
C01429=1124.892,284.730,-74.288,-178.104,10.289,149.548
C01430=1124.887,284.978,-74.319,-178.100,10.291,149.548
C01431=1124.884,285.226,-74.349,-178.098,10.294,149.547
C01432=1124.880,285.475,-74.380,-178.095,10.297,149.547
C01433=1124.875,285.723,-74.411,-178.092,10.298,149.547
C01434=1124.871,285.970,-74.441,-178.089,10.301,149.547
C01435=1124.867,286.219,-74.472,-178.086,10.304,149.547
C01436=1124.862,286.467,-74.503,-178.083,10.306,149.547
C01437=1124.859,286.714,-74.533,-178.079,10.309,149.546
C01438=1124.855,286.963,-74.564,-178.076,10.312,149.546
C01439=1124.850,287.211,-74.595,-178.073,10.314,149.546
C01440=1124.846,287.459,-74.625,-178.070,10.317,149.546
C01441=1124.842,287.707,-74.656,-178.067,10.320,149.546
C01442=1124.838,287.955,-74.688,-178.064,10.322,149.545
C01443=1124.833,288.203,-74.718,-178.062,10.324,149.545
C01444=1124.830,288.451,-74.749,-178.058,10.326,149.545
C01445=1124.825,288.699,-74.780,-178.055,10.329,149.545
C01446=1124.821,288.948,-74.811,-178.052,10.332,149.545
C01447=1124.817,289.196,-74.842,-178.049,10.334,149.545
C01448=1124.813,289.443,-74.872,-178.046,10.337,149.544
C01449=1124.809,289.691,-74.904,-178.043,10.339,149.544
C01450=1124.804,289.939,-74.934,-178.040,10.342,149.544
C01451=1124.800,290.188,-74.965,-178.036,10.345,149.544
C01452=1124.796,290.435,-74.997,-178.034,10.347,149.544
C01453=1124.793,290.684,-75.027,-178.031,10.349,149.544
C01454=1124.788,290.932,-75.058,-178.028,10.352,149.543
C01455=1124.784,291.180,-75.089,-178.025,10.354,149.543
C01456=1124.780,291.428,-75.121,-178.022,10.357,149.543
C01457=1124.775,291.676,-75.152,-178.018,10.359,149.543
C01458=1124.771,291.924,-75.183,-178.015,10.362,149.543
C01459=1124.768,292.171,-75.214,-178.012,10.365,149.542
C01460=1124.764,292.420,-75.245,-178.009,10.367,149.542
C01461=1124.759,292.668,-75.276,-178.006,10.370,149.542
C01462=1124.755,292.916,-75.307,-178.003,10.373,149.542
C01463=1124.751,293.164,-75.338,-178.000,10.375,149.542
C01464=1124.747,293.412,-75.370,-177.997,10.377,149.542
C01465=1124.743,293.625,-75.396,-177.994,10.380,149.542
C01466=1124.740,293.839,-75.423,-177.992,10.382,149.541
C01467=1124.736,294.051,-75.451,-177.989,10.384,149.541
C01468=1124.733,294.264,-75.476,-177.986,10.386,149.541
C01469=1124.729,294.478,-75.503,-177.984,10.388,149.541
C01470=1124.726,294.690,-75.531,-177.981,10.391,149.541
C01471=1124.722,294.904,-75.557,-177.978,10.393,149.541
C01472=1124.719,295.117,-75.585,-177.976,10.395,149.540
C01473=1124.715,295.365,-75.616,-177.973,10.397,149.540
C01474=1124.710,295.613,-75.647,-177.970,10.400,149.540
C01475=1124.706,295.861,-75.678,-177.966,10.402,149.540
C01476=1124.702,296.109,-75.710,-177.963,10.405,149.540
C01477=1124.698,296.357,-75.741,-177.960,10.407,149.539
C01478=1124.694,296.605,-75.773,-177.957,10.410,149.539
C01479=1124.690,296.853,-75.804,-177.954,10.413,149.539
C01480=1124.686,297.101,-75.835,-177.951,10.415,149.539
C01481=1124.682,297.349,-75.867,-177.948,10.418,149.539
C01482=1124.678,297.597,-75.899,-177.945,10.420,149.539
C01483=1124.673,297.845,-75.930,-177.942,10.423,149.539
C01484=1124.669,298.093,-75.962,-177.939,10.425,149.538
C01485=1124.665,298.341,-75.994,-177.936,10.428,149.538
C01486=1124.661,298.589,-76.025,-177.933,10.430,149.538
C01487=1124.657,298.837,-76.056,-177.930,10.433,149.538
C01488=1124.653,299.084,-76.088,-177.927,10.435,149.538
C01489=1124.649,299.332,-76.120,-177.923,10.438,149.537
C01490=1124.645,299.581,-76.151,-177.920,10.441,149.537
C01491=1124.640,299.828,-76.182,-177.917,10.443,149.537
C01492=1124.636,300.077,-76.215,-177.914,10.446,149.537
C01493=1124.632,300.324,-76.246,-177.911,10.447,149.537
C01494=1124.628,300.572,-76.278,-177.908,10.450,149.536
C01495=1124.624,300.821,-76.309,-177.905,10.453,149.536
C01496=1124.620,301.068,-76.341,-177.902,10.455,149.536
C01497=1124.615,301.317,-76.373,-177.899,10.458,149.536
C01498=1124.612,301.565,-76.405,-177.896,10.461,149.536
C01499=1124.607,301.812,-76.436,-177.892,10.463,149.535
C01500=1124.604,302.060,-76.468,-177.890,10.466,149.535
C01501=1124.599,302.308,-76.501,-177.886,10.468,149.535
C01502=1124.595,302.556,-76.532,-177.883,10.471,149.535
C01503=1124.591,302.804,-76.564,-177.880,10.473,149.535
C01504=1124.587,303.052,-76.595,-177.877,10.476,149.535
C01505=1124.582,303.300,-76.627,-177.874,10.479,149.534
C01506=1124.578,303.548,-76.659,-177.871,10.481,149.534
C01507=1124.575,303.796,-76.691,-177.868,10.483,149.534
C01508=1124.570,304.044,-76.723,-177.865,10.486,149.534
C01509=1124.566,304.292,-76.755,-177.862,10.488,149.534
C01510=1124.562,304.539,-76.787,-177.859,10.491,149.534
C01511=1124.558,304.787,-76.820,-177.856,10.493,149.533
C01512=1124.554,305.035,-76.851,-177.852,10.496,149.533
C01513=1124.550,305.283,-76.883,-177.849,10.499,149.533
C01514=1124.546,305.531,-76.916,-177.846,10.501,149.533
C01515=1124.542,305.779,-76.947,-177.843,10.504,149.533
C01516=1124.538,306.027,-76.979,-177.840,10.506,149.532
C01517=1124.533,306.275,-77.011,-177.837,10.509,149.532
C01518=1124.529,306.523,-77.043,-177.834,10.511,149.532
C01519=1124.525,306.771,-77.076,-177.831,10.513,149.532
C01520=1124.521,307.018,-77.108,-177.828,10.516,149.532
C01521=1124.518,307.231,-77.135,-177.825,10.519,149.532
C01522=1124.514,307.445,-77.164,-177.822,10.520,149.531
C01523=1124.510,307.657,-77.191,-177.820,10.522,149.531
C01524=1124.507,307.870,-77.218,-177.817,10.525,149.531
C01525=1124.503,308.084,-77.247,-177.814,10.527,149.531
C01526=1124.500,308.296,-77.274,-177.811,10.529,149.531
C01527=1124.497,308.510,-77.301,-177.809,10.531,149.531
C01528=1124.493,308.723,-77.330,-177.806,10.533,149.530
C01529=1124.489,308.970,-77.361,-177.803,10.536,149.530
C01530=1124.484,309.218,-77.394,-177.800,10.538,149.530
C01531=1124.481,309.466,-77.426,-177.797,10.541,149.530
C01532=1124.476,309.715,-77.458,-177.794,10.544,149.530
C01533=1124.473,309.962,-77.491,-177.791,10.546,149.530
C01534=1124.468,310.210,-77.523,-177.788,10.549,149.529
C01535=1124.465,310.458,-77.556,-177.784,10.551,149.529
C01536=1124.460,310.705,-77.588,-177.781,10.554,149.529
C01537=1124.456,310.953,-77.620,-177.778,10.556,149.529
C01538=1124.452,311.201,-77.653,-177.775,10.559,149.529
C01539=1124.448,311.449,-77.685,-177.772,10.561,149.528
C01540=1124.444,311.697,-77.718,-177.769,10.564,149.528
C01541=1124.441,311.945,-77.750,-177.766,10.566,149.528
C01542=1124.436,312.193,-77.783,-177.763,10.568,149.528
C01543=1124.432,312.441,-77.816,-177.760,10.571,149.528
C01544=1124.428,312.688,-77.848,-177.756,10.574,149.528
C01545=1124.424,312.936,-77.880,-177.754,10.576,149.528
C01546=1124.420,313.184,-77.913,-177.750,10.579,149.527
C01547=1124.416,313.432,-77.945,-177.747,10.581,149.527
C01548=1124.412,313.680,-77.978,-177.744,10.584,149.527
C01549=1124.408,313.928,-78.010,-177.741,10.587,149.527
C01550=1124.404,314.175,-78.043,-177.738,10.589,149.527
C01551=1124.400,314.423,-78.076,-177.734,10.592,149.526
C01552=1124.396,314.671,-78.108,-177.731,10.594,149.526
C01553=1124.392,314.919,-78.141,-177.729,10.596,149.526
C01554=1124.388,315.167,-78.175,-177.725,10.599,149.526
C01555=1124.384,315.415,-78.206,-177.722,10.601,149.526
C01556=1124.380,315.662,-78.240,-177.719,10.604,149.525
C01557=1124.376,315.910,-78.273,-177.716,10.606,149.525
C01558=1124.371,316.158,-78.305,-177.713,10.609,149.525
C01559=1124.368,316.406,-78.338,-177.710,10.611,149.525
C01560=1124.364,316.654,-78.371,-177.707,10.614,149.525
C01561=1124.359,316.901,-78.404,-177.703,10.617,149.525
C01562=1124.356,317.149,-78.436,-177.700,10.619,149.524
C01563=1124.352,317.397,-78.469,-177.697,10.622,149.524
C01564=1124.347,317.645,-78.502,-177.694,10.624,149.524
C01565=1124.343,317.893,-78.535,-177.691,10.627,149.524
C01566=1124.339,318.140,-78.569,-177.687,10.630,149.524
C01567=1124.335,318.388,-78.600,-177.684,10.632,149.523
C01568=1124.331,318.636,-78.634,-177.682,10.634,149.523
C01569=1124.327,318.884,-78.667,-177.679,10.636,149.523
C01570=1124.323,319.132,-78.700,-177.675,10.639,149.523
C01571=1124.319,319.379,-78.733,-177.672,10.642,149.523
C01572=1124.316,319.627,-78.766,-177.669,10.644,149.522
C01573=1124.311,319.874,-78.799,-177.666,10.647,149.522
C01574=1124.307,320.122,-78.832,-177.663,10.649,149.522
C01575=1124.303,320.370,-78.865,-177.659,10.652,149.522
C01576=1124.299,320.618,-78.898,-177.656,10.655,149.522
C01577=1124.295,320.831,-78.926,-177.654,10.656,149.522
C01578=1124.292,321.044,-78.955,-177.651,10.659,149.521
C01579=1124.289,321.257,-78.984,-177.648,10.661,149.521
C01580=1124.285,321.469,-79.012,-177.646,10.663,149.521
C01581=1124.282,321.683,-79.040,-177.643,10.665,149.521
C01582=1124.279,321.895,-79.069,-177.640,10.667,149.521
C01583=1124.275,322.108,-79.098,-177.637,10.670,149.521
C01584=1124.272,322.321,-79.126,-177.635,10.672,149.520
C01585=1124.268,322.569,-79.159,-177.632,10.674,149.520
C01586=1124.264,322.816,-79.192,-177.628,10.677,149.520
C01587=1124.260,323.064,-79.226,-177.625,10.679,149.520
C01588=1124.256,323.312,-79.259,-177.622,10.682,149.520
C01589=1124.252,323.560,-79.292,-177.619,10.684,149.520
C01590=1124.248,323.807,-79.325,-177.615,10.687,149.519
C01591=1124.244,324.055,-79.359,-177.613,10.690,149.519
C01592=1124.240,324.303,-79.392,-177.610,10.691,149.519
C01593=1124.236,324.551,-79.426,-177.607,10.694,149.519
C01594=1124.232,324.798,-79.459,-177.604,10.697,149.519
C01595=1124.228,325.046,-79.492,-177.600,10.699,149.518
C01596=1124.224,325.293,-79.526,-177.597,10.701,149.518
C01597=1124.220,325.542,-79.559,-177.594,10.704,149.518
C01598=1124.216,325.790,-79.593,-177.591,10.707,149.518
C01599=1124.211,326.037,-79.626,-177.587,10.709,149.518
C01600=1124.208,326.284,-79.660,-177.584,10.712,149.518
C01601=1124.203,326.532,-79.693,-177.581,10.714,149.517
C01602=1124.200,326.781,-79.727,-177.578,10.717,149.517
C01603=1124.196,327.028,-79.761,-177.574,10.719,149.517
C01604=1124.192,327.275,-79.794,-177.572,10.722,149.517
C01605=1124.188,327.523,-79.827,-177.568,10.724,149.516
C01606=1124.184,327.770,-79.861,-177.565,10.727,149.516
C01607=1124.180,328.019,-79.895,-177.562,10.730,149.516
C01608=1124.176,328.266,-79.929,-177.559,10.731,149.516
C01609=1124.172,328.514,-79.962,-177.556,10.734,149.516
C01610=1124.168,328.762,-79.995,-177.553,10.737,149.516
C01611=1124.164,329.009,-80.029,-177.550,10.739,149.515
C01612=1124.159,329.257,-80.063,-177.546,10.741,149.515
C01613=1124.156,329.505,-80.097,-177.543,10.744,149.515
C01614=1124.152,329.752,-80.130,-177.540,10.747,149.515
C01615=1124.148,330.000,-80.164,-177.537,10.749,149.515
C01616=1124.144,330.248,-80.197,-177.534,10.752,149.514
C01617=1124.140,330.495,-80.232,-177.531,10.754,149.514
C01618=1124.136,330.744,-80.265,-177.527,10.757,149.514
C01619=1124.132,330.991,-80.299,-177.524,10.759,149.514
C01620=1124.128,331.238,-80.333,-177.521,10.762,149.514
C01621=1124.124,331.487,-80.367,-177.518,10.764,149.513
C01622=1124.120,331.734,-80.401,-177.514,10.767,149.513
C01623=1124.116,331.981,-80.434,-177.511,10.769,149.513
C01624=1124.112,332.230,-80.469,-177.509,10.771,149.513
C01625=1124.108,332.477,-80.503,-177.505,10.774,149.513
C01626=1124.104,332.724,-80.536,-177.502,10.776,149.512
C01627=1124.100,332.973,-80.571,-177.499,10.779,149.512
C01628=1124.096,333.220,-80.605,-177.496,10.781,149.512
C01629=1124.092,333.467,-80.638,-177.493,10.784,149.512
C01630=1124.088,333.716,-80.673,-177.489,10.786,149.512
C01631=1124.084,333.963,-80.707,-177.486,10.789,149.511
C01632=1124.081,334.210,-80.741,-177.483,10.792,149.511
C01633=1124.077,334.423,-80.770,-177.480,10.793,149.511
C01634=1124.074,334.636,-80.799,-177.477,10.796,149.511
C01635=1124.070,334.849,-80.829,-177.475,10.798,149.511
C01636=1124.067,335.062,-80.858,-177.472,10.801,149.511
C01637=1124.064,335.274,-80.887,-177.469,10.802,149.510
C01638=1124.060,335.487,-80.916,-177.467,10.804,149.510
C01639=1124.057,335.699,-80.946,-177.464,10.807,149.510
C01640=1124.053,335.912,-80.975,-177.461,10.809,149.510
C01641=1124.049,336.160,-81.010,-177.458,10.811,149.510
C01642=1124.045,336.407,-81.044,-177.455,10.814,149.510
C01643=1124.042,336.655,-81.078,-177.451,10.816,149.509
C01644=1124.038,336.902,-81.112,-177.448,10.819,149.509
C01645=1124.034,337.149,-81.146,-177.445,10.821,149.509
C01646=1124.030,337.398,-81.181,-177.442,10.824,149.509
C01647=1124.026,337.645,-81.214,-177.438,10.826,149.509
C01648=1124.022,337.893,-81.249,-177.435,10.829,149.508
C01649=1124.018,338.141,-81.283,-177.432,10.831,149.508
C01650=1124.014,338.389,-81.318,-177.429,10.834,149.508
C01651=1124.010,338.636,-81.351,-177.426,10.836,149.508
C01652=1124.006,338.884,-81.386,-177.423,10.838,149.507
C01653=1124.002,339.131,-81.421,-177.420,10.841,149.507
C01654=1123.999,339.379,-81.456,-177.417,10.843,149.507
C01655=1123.994,339.626,-81.490,-177.413,10.846,149.507
C01656=1123.991,339.874,-81.524,-177.410,10.848,149.507
C01657=1123.986,340.121,-81.559,-177.407,10.851,149.506
C01658=1123.982,340.369,-81.594,-177.404,10.853,149.506
C01659=1123.978,340.616,-81.628,-177.400,10.856,149.506
C01660=1123.974,340.865,-81.662,-177.397,10.858,149.506
C01661=1123.971,341.112,-81.696,-177.394,10.861,149.506
C01662=1123.967,341.360,-81.731,-177.391,10.863,149.506
C01663=1123.962,341.607,-81.766,-177.388,10.866,149.505
C01664=1123.959,341.854,-81.801,-177.384,10.868,149.505
C01665=1123.955,342.102,-81.835,-177.381,10.871,149.505
C01666=1123.951,342.350,-81.870,-177.378,10.873,149.505
C01667=1123.947,342.597,-81.904,-177.374,10.876,149.505
C01668=1123.943,342.845,-81.939,-177.371,10.878,149.504
C01669=1123.939,343.092,-81.974,-177.369,10.880,149.504
C01670=1123.935,343.340,-82.009,-177.365,10.883,149.504
C01671=1123.931,343.587,-82.043,-177.362,10.885,149.504
C01672=1123.927,343.835,-82.078,-177.359,10.888,149.504
C01673=1123.923,344.083,-82.113,-177.355,10.890,149.503
C01674=1123.919,344.330,-82.147,-177.353,10.893,149.503
C01675=1123.916,344.577,-82.182,-177.349,10.895,149.503
C01676=1123.911,344.825,-82.217,-177.346,10.898,149.503
C01677=1123.907,345.072,-82.252,-177.343,10.900,149.503
C01678=1123.903,345.320,-82.287,-177.339,10.903,149.502
C01679=1123.900,345.568,-82.321,-177.336,10.905,149.502
C01680=1123.896,345.815,-82.357,-177.333,10.908,149.502
C01681=1123.891,346.062,-82.391,-177.330,10.910,149.502
C01682=1123.888,346.310,-82.427,-177.326,10.913,149.502
C01683=1123.884,346.558,-82.461,-177.323,10.915,149.501
C01684=1123.880,346.805,-82.496,-177.320,10.918,149.501
C01685=1123.876,347.053,-82.531,-177.317,10.920,149.501
C01686=1123.873,347.300,-82.566,-177.313,10.923,149.501
C01687=1123.868,347.548,-82.601,-177.311,10.925,149.501
C01688=1123.864,347.795,-82.636,-177.308,10.927,149.500
C01689=1123.861,348.007,-82.666,-177.304,10.930,149.500
C01690=1123.858,348.221,-82.697,-177.302,10.931,149.500
C01691=1123.855,348.433,-82.726,-177.299,10.934,149.500
C01692=1123.851,348.645,-82.756,-177.296,10.936,149.500
C01693=1123.848,348.858,-82.786,-177.294,10.938,149.499
C01694=1123.844,349.071,-82.816,-177.290,10.940,149.499
C01695=1123.841,349.283,-82.847,-177.288,10.942,149.499
C01696=1123.838,349.496,-82.877,-177.285,10.945,149.499
C01697=1123.833,349.743,-82.912,-177.282,10.947,149.499
C01698=1123.830,349.991,-82.947,-177.278,10.950,149.498
C01699=1123.826,350.238,-82.983,-177.274,10.952,149.498
C01700=1123.822,350.486,-83.018,-177.271,10.955,149.498
C01701=1123.818,350.733,-83.053,-177.267,10.957,149.498
C01702=1123.814,350.981,-83.088,-177.264,10.960,149.497
C01703=1123.810,351.228,-83.124,-177.261,10.962,149.497
C01704=1123.806,351.476,-83.159,-177.257,10.966,149.497
C01705=1123.802,351.723,-83.194,-177.253,10.968,149.497
C01706=1123.798,351.971,-83.230,-177.250,10.970,149.496
C01707=1123.795,352.218,-83.265,-177.246,10.973,149.496
C01708=1123.791,352.466,-83.301,-177.242,10.976,149.496
C01709=1123.787,352.712,-83.336,-177.239,10.978,149.496
C01710=1123.783,352.961,-83.371,-177.235,10.981,149.495
C01711=1123.779,353.208,-83.406,-177.232,10.983,149.495
C01712=1123.776,353.456,-83.442,-177.229,10.985,149.495
C01713=1123.772,353.703,-83.477,-177.225,10.989,149.495
C01714=1123.768,353.950,-83.513,-177.222,10.991,149.494
C01715=1123.764,354.197,-83.548,-177.218,10.993,149.494
C01716=1123.760,354.445,-83.584,-177.214,10.996,149.494
C01717=1123.757,354.692,-83.619,-177.211,10.998,149.494
C01718=1123.753,354.940,-83.655,-177.208,11.001,149.493
C01719=1123.749,355.188,-83.691,-177.204,11.004,149.493
C01720=1123.744,355.435,-83.726,-177.200,11.006,149.493
C01721=1123.741,355.682,-83.762,-177.197,11.009,149.493
C01722=1123.737,355.930,-83.797,-177.194,11.011,149.492
C01723=1123.733,356.177,-83.833,-177.190,11.013,149.492
C01724=1123.730,356.425,-83.868,-177.187,11.016,149.492
C01725=1123.725,356.672,-83.904,-177.183,11.018,149.492
C01726=1123.722,356.920,-83.940,-177.180,11.021,149.491
C01727=1123.717,357.167,-83.975,-177.176,11.024,149.491
C01728=1123.714,357.413,-84.011,-177.172,11.026,149.491
C01729=1123.710,357.661,-84.047,-177.169,11.028,149.490
C01730=1123.706,357.909,-84.083,-177.166,11.031,149.490
C01731=1123.702,358.156,-84.119,-177.162,11.033,149.490
C01732=1123.699,358.404,-84.154,-177.159,11.035,149.490
C01733=1123.695,358.651,-84.190,-177.155,11.038,149.489
C01734=1123.691,358.898,-84.227,-177.152,11.040,149.489
C01735=1123.687,359.146,-84.262,-177.149,11.043,149.489
C01736=1123.684,359.394,-84.298,-177.145,11.045,149.489
C01737=1123.680,359.640,-84.334,-177.142,11.047,149.488
C01738=1123.676,359.888,-84.370,-177.138,11.050,149.488
C01739=1123.672,360.136,-84.406,-177.135,11.052,149.488
C01740=1123.669,360.383,-84.442,-177.131,11.055,149.488
C01741=1123.664,360.630,-84.478,-177.128,11.057,149.487
C01742=1123.661,360.878,-84.514,-177.125,11.059,149.487
C01743=1123.657,361.125,-84.550,-177.122,11.062,149.487
C01744=1123.653,361.373,-84.586,-177.118,11.064,149.487
C01745=1123.650,361.584,-84.616,-177.115,11.067,149.486
C01746=1123.647,361.797,-84.648,-177.112,11.069,149.486
C01747=1123.643,362.009,-84.678,-177.110,11.070,149.486
C01748=1123.640,362.222,-84.709,-177.106,11.073,149.486
C01749=1123.637,362.435,-84.740,-177.104,11.074,149.485
C01750=1123.633,362.647,-84.771,-177.100,11.077,149.485
C01751=1123.630,362.859,-84.802,-177.098,11.079,149.485
C01752=1123.627,363.071,-84.833,-177.094,11.081,149.485
C01753=1123.623,363.318,-84.870,-177.092,11.083,149.485
C01754=1123.619,363.566,-84.906,-177.088,11.085,149.484
C01755=1123.616,363.814,-84.942,-177.085,11.088,149.484
C01756=1123.612,364.061,-84.979,-177.082,11.090,149.484
C01757=1123.608,364.308,-85.015,-177.078,11.092,149.483
C01758=1123.605,364.556,-85.050,-177.075,11.095,149.483
C01759=1123.601,364.803,-85.087,-177.071,11.097,149.483
C01760=1123.597,365.050,-85.123,-177.068,11.100,149.483
C01761=1123.593,365.298,-85.160,-177.065,11.102,149.483
C01762=1123.589,365.544,-85.196,-177.062,11.105,149.482
C01763=1123.585,365.792,-85.232,-177.058,11.107,149.482
C01764=1123.582,366.039,-85.268,-177.055,11.109,149.482
C01765=1123.578,366.286,-85.305,-177.051,11.112,149.482
C01766=1123.573,366.534,-85.341,-177.049,11.113,149.481
C01767=1123.570,366.781,-85.378,-177.045,11.116,149.481
C01768=1123.566,367.028,-85.414,-177.042,11.118,149.481
C01769=1123.562,367.309,-85.456,-177.038,11.121,149.481
C01770=1123.558,367.589,-85.497,-177.034,11.124,149.480
C01771=1123.553,367.870,-85.539,-177.031,11.126,149.480
C01772=1123.549,368.150,-85.580,-177.027,11.129,149.480
C01773=1123.546,368.397,-85.616,-177.023,11.132,149.480
C01774=1123.541,368.644,-85.653,-177.020,11.134,149.479
C01775=1123.537,368.891,-85.690,-177.017,11.136,149.479
C01776=1123.534,369.138,-85.726,-177.014,11.138,149.479
C01777=1123.530,369.387,-85.762,-177.011,11.141,149.479
C01778=1123.526,369.634,-85.799,-177.008,11.143,149.479
C01779=1123.523,369.881,-85.836,-177.004,11.146,149.478
C01780=1123.519,370.128,-85.872,-177.001,11.148,149.478
C01781=1123.515,370.375,-85.909,-176.998,11.151,149.478
C01782=1123.511,370.622,-85.946,-176.995,11.152,149.478
C01783=1123.508,370.870,-85.983,-176.992,11.155,149.477
C01784=1123.504,371.117,-86.020,-176.988,11.157,149.477
C01785=1123.500,371.364,-86.056,-176.985,11.160,149.477
C01786=1123.496,371.611,-86.093,-176.982,11.162,149.477
C01787=1123.492,371.859,-86.130,-176.978,11.165,149.477
C01788=1123.489,372.106,-86.167,-176.976,11.166,149.476
C01789=1123.485,372.353,-86.203,-176.972,11.169,149.476
C01790=1123.481,372.600,-86.240,-176.969,11.171,149.476
C01791=1123.477,372.848,-86.277,-176.966,11.174,149.476
C01792=1123.474,373.096,-86.314,-176.963,11.176,149.476
C01793=1123.470,373.342,-86.350,-176.960,11.178,149.475
C01794=1123.466,373.590,-86.387,-176.957,11.181,149.475
C01795=1123.462,373.837,-86.424,-176.954,11.183,149.475
C01796=1123.458,374.085,-86.461,-176.950,11.186,149.475
C01797=1123.455,374.331,-86.498,-176.947,11.188,149.475
C01798=1123.451,374.578,-86.535,-176.944,11.190,149.474
C01799=1123.447,374.825,-86.572,-176.941,11.193,149.474
C01800=1123.444,375.073,-86.609,-176.938,11.195,149.474
C01801=1123.437,375.465,-86.667,-176.933,11.199,149.474
C01802=1123.432,375.856,-86.727,-176.928,11.203,149.474
C01803=1123.425,376.248,-86.785,-176.923,11.206,149.473
C01804=1123.419,376.639,-86.844,-176.918,11.210,149.473
C01805=1123.415,376.886,-86.881,-176.916,11.213,149.473
C01806=1123.412,377.133,-86.919,-176.913,11.215,149.473
C01807=1123.409,377.380,-86.955,-176.910,11.217,149.473
C01808=1123.405,377.628,-86.992,-176.907,11.220,149.473
C01809=1123.401,377.875,-87.029,-176.903,11.223,149.472
C01810=1123.397,378.122,-87.067,-176.901,11.224,149.472
C01811=1123.393,378.369,-87.103,-176.898,11.227,149.472
C01812=1123.390,378.616,-87.141,-176.895,11.230,149.472
C01813=1123.386,378.864,-87.178,-176.891,11.232,149.472
C01814=1123.382,379.111,-87.215,-176.889,11.234,149.472
C01815=1123.379,379.358,-87.253,-176.886,11.237,149.471
C01816=1123.375,379.605,-87.290,-176.883,11.239,149.471
C01817=1123.372,379.853,-87.328,-176.880,11.242,149.471
C01818=1123.367,380.100,-87.365,-176.877,11.244,149.471
C01819=1123.364,380.346,-87.402,-176.874,11.246,149.471
C01820=1123.360,380.594,-87.440,-176.871,11.249,149.471
